  MoveL 3325 to (-39.23, 44.12, 59.84) mm, rotated rx -180 ry 0 rz 180 deg; joints [-136.898, -56.439, -94.12, 47.06, 68.969, -21.09]
  MoveL 3326 to (-39.23, 44.12, 59.84) mm, rotated rx -180 ry 0 rz 180 deg; joints [-136.898, -56.439, -94.12, 47.06, 68.969, -21.09]
  Call Extruder(64.50294)
  MoveL 3327 to (-39.1, 43.83, 59.84) mm, rotated rx 180 ry 0 rz -180 deg; joints [-136.946, -56.434, -94.139, 47.008, 68.961, -21.062]
  MoveL 3328 to (-39.1, 43.83, 59.84) mm, rotated rx 180 ry 0 rz -180 deg; joints [-136.946, -56.434, -94.139, 47.008, 68.961, -21.062]
  Call Extruder(64.66063)
  MoveL 3329 to (-39, 43.58, 59.84) mm, rotated rx -180 ry 0 rz -180 deg; joints [-136.988, -56.429, -94.155, 46.963, 68.953, -21.038]
  MoveL 3330 to (-39, 43.58, 59.84) mm, rotated rx -180 ry 0 rz -180 deg; joints [-136.988, -56.429, -94.155, 46.963, 68.953, -21.038]
  Call Extruder(64.81891)
  MoveL 3331 to (-38.89, 43.34, 59.84) mm, rotated rx 180 ry 0 rz 180 deg; joints [-137.029, -56.425, -94.17, 46.919, 68.946, -21.015]
  MoveL 3332 to (-38.89, 43.34, 59.84) mm, rotated rx 180 ry 0 rz 180 deg; joints [-137.029, -56.425, -94.17, 46.919, 68.946, -21.015]
  Call Extruder(65.00094)
  MoveL 3333 to (-38.75, 43.06, 59.84) mm, rotated rx 180 ry 0 rz -180 deg; joints [-137.078, -56.421, -94.184, 46.867, 68.935, -20.989]
  MoveL 3334 to (-38.75, 43.06, 59.84) mm, rotated rx 180 ry 0 rz -180 deg; joints [-137.078, -56.421, -94.184, 46.867, 68.935, -20.989]
  Call Extruder(65.20749)
  MoveL 3335 to (-38.57, 42.75, 59.84) mm, rotated rx -180 ry 0 rz -180 deg; joints [-137.135, -56.417, -94.197, 46.808, 68.921, -20.961]
  MoveL 3336 to (-38.57, 42.75, 59.84) mm, rotated rx -180 ry 0 rz -180 deg; joints [-137.135, -56.417, -94.197, 46.808, 68.921, -20.961]
  Call Extruder(65.41482)
  MoveL 3337 to (-38.4, 42.45, 59.84) mm, rotated rx 180 ry 0 rz -180 deg; joints [-137.191, -56.413, -94.21, 46.749, 68.908, -20.934]
  MoveL 3338 to (-38.4, 42.45, 59.84) mm, rotated rx 180 ry 0 rz -180 deg; joints [-137.191, -56.413, -94.21, 46.749, 68.908, -20.934]
  Call Extruder(65.62294)
  MoveL 3339 to (-38.22, 42.15, 59.84) mm, rotated rx 180 ry 0 rz 180 deg; joints [-137.247, -56.41, -94.223, 46.69, 68.894, -20.906]
  MoveL 3340 to (-38.22, 42.15, 59.84) mm, rotated rx 180 ry 0 rz 180 deg; joints [-137.247, -56.41, -94.223, 46.69, 68.894, -20.906]
  Call Extruder(65.74065)
  MoveL 3341 to (-38.12, 41.97, 59.84) mm, rotated rx -180 ry 0 rz -180 deg; joints [-137.279, -56.408, -94.231, 46.657, 68.886, -20.891]
  MoveL 3342 to (-38.12, 41.97, 59.84) mm, rotated rx -180 ry 0 rz -180 deg; joints [-137.279, -56.408, -94.231, 46.657, 68.886, -20.891]
  Call Extruder(66.07350)
  MoveL 3343 to (-37.79, 41.52, 59.84) mm, rotated rx 180 ry 0 rz 180 deg; joints [-137.37, -56.405, -94.241, 46.564, 68.859, -20.852]
  MoveL 3344 to (-37.79, 41.52, 59.84) mm, rotated rx 180 ry 0 rz 180 deg; joints [-137.37, -56.405, -94.241, 46.564, 68.859, -20.852]
  Call Extruder(66.40753)
  MoveL 3345 to (-37.47, 41.07, 59.84) mm, rotated rx 180 ry 0 rz 180 deg; joints [-137.461, -56.402, -94.252, 46.47, 68.832, -20.813]
  MoveL 3346 to (-37.47, 41.07, 59.84) mm, rotated rx 180 ry 0 rz 180 deg; joints [-137.461, -56.402, -94.252, 46.47, 68.832, -20.813]
  Call Extruder(66.57512)
  MoveL 3347 to (-37.3, 40.85, 59.84) mm, rotated rx 180 ry 0 rz 180 deg; joints [-137.506, -56.4, -94.257, 46.424, 68.819, -20.794]
  Call Extruder(67.40443)
  MoveL 3348 to (-36.39, 39.81, 59.84) mm, rotated rx 180 ry 0 rz -180 deg; joints [-137.733, -56.399, -94.262, 46.195, 68.74, -20.709]
  Call Extruder(68.03550)
  MoveL 3349 to (-35.6, 39.11, 59.84) mm, rotated rx 180 ry 0 rz 180 deg; joints [-137.904, -56.404, -94.243, 46.027, 68.67, -20.657]
  MoveL 3350 to (-35.6, 39.11, 59.84) mm, rotated rx 180 ry 0 rz 180 deg; joints [-137.904, -56.404, -94.243, 46.027, 68.67, -20.657]
  Call Extruder(68.23307)
  MoveL 3351 to (-35.35, 38.9, 59.84) mm, rotated rx 180 ry 0 rz -180 deg; joints [-137.958, -56.406, -94.235, 45.974, 68.648, -20.641]
  Call Extruder(68.56709)
  MoveL 3352 to (-34.9, 38.57, 59.84) mm, rotated rx 180 ry 0 rz -180 deg; joints [-138.048, -56.412, -94.216, 45.888, 68.606, -20.619]
  MoveL 3353 to (-34.9, 38.57, 59.84) mm, rotated rx 180 ry 0 rz -180 deg; joints [-138.048, -56.412, -94.216, 45.888, 68.606, -20.619]
  Call Extruder(68.89992)
  MoveL 3354 to (-34.45, 38.24, 59.84) mm, rotated rx -180 ry 0 rz 180 deg; joints [-138.137, -56.417, -94.196, 45.802, 68.565, -20.597]
  MoveL 3355 to (-34.45, 38.24, 59.84) mm, rotated rx -180 ry 0 rz 180 deg; joints [-138.137, -56.417, -94.196, 45.802, 68.565, -20.597]
  Call Extruder(69.07917)
  MoveL 3356 to (-34.21, 38.07, 59.84) mm, rotated rx 180 ry 0 rz 180 deg; joints [-138.185, -56.42, -94.185, 45.756, 68.543, -20.586]
  MoveL 3357 to (-34.21, 38.07, 59.84) mm, rotated rx 180 ry 0 rz 180 deg; joints [-138.185, -56.42, -94.185, 45.756, 68.543, -20.586]
  Call Extruder(69.28728)
  MoveL 3358 to (-33.9, 37.89, 59.84) mm, rotated rx 180 ry 0 rz -180 deg; joints [-138.24, -56.426, -94.167, 45.705, 68.514, -20.576]
  MoveL 3359 to (-33.9, 37.89, 59.84) mm, rotated rx 180 ry 0 rz -180 deg; joints [-138.24, -56.426, -94.167, 45.705, 68.514, -20.576]
  Call Extruder(69.49461)
  MoveL 3360 to (-33.6, 37.71, 59.84) mm, rotated rx -180 ry 0 rz -180 deg; joints [-138.295, -56.431, -94.149, 45.653, 68.486, -20.566]
  MoveL 3361 to (-33.6, 37.71, 59.84) mm, rotated rx -180 ry 0 rz -180 deg; joints [-138.295, -56.431, -94.149, 45.653, 68.486, -20.566]
  Call Extruder(69.70116)
  MoveL 3362 to (-33.29, 37.54, 59.84) mm, rotated rx 180 ry 0 rz 180 deg; joints [-138.349, -56.436, -94.13, 45.602, 68.458, -20.556]
  MoveL 3363 to (-33.29, 37.54, 59.84) mm, rotated rx 180 ry 0 rz 180 deg; joints [-138.349, -56.436, -94.13, 45.602, 68.458, -20.556]
  Call Extruder(69.90693)
  MoveL 3364 to (-32.99, 37.36, 59.84) mm, rotated rx 180 ry 0 rz 180 deg; joints [-138.404, -56.441, -94.112, 45.551, 68.429, -20.546]
  MoveL 3365 to (-32.99, 37.36, 59.84) mm, rotated rx 180 ry 0 rz 180 deg; joints [-138.404, -56.441, -94.112, 45.551, 68.429, -20.546]
  Call Extruder(70.06523)
  MoveL 3366 to (-32.74, 37.26, 59.84) mm, rotated rx -180 ry 0 rz 180 deg; joints [-138.444, -56.447, -94.092, 45.514, 68.405, -20.541]
  MoveL 3367 to (-32.74, 37.26, 59.84) mm, rotated rx -180 ry 0 rz 180 deg; joints [-138.444, -56.447, -94.092, 45.514, 68.405, -20.541]
  Call Extruder(70.22293)
  MoveL 3368 to (-32.49, 37.15, 59.84) mm, rotated rx 180 ry 0 rz 180 deg; joints [-138.484, -56.452, -94.073, 45.478, 68.381, -20.537]
  MoveL 3369 to (-32.49, 37.15, 59.84) mm, rotated rx 180 ry 0 rz 180 deg; joints [-138.484, -56.452, -94.073, 45.478, 68.381, -20.537]
  Call Extruder(70.39301)
  MoveL 3370 to (-32.22, 37.03, 59.84) mm, rotated rx -180 ry 0 rz 180 deg; joints [-138.527, -56.459, -94.051, 45.439, 68.356, -20.533]
  MoveL 3371 to (-32.22, 37.03, 59.84) mm, rotated rx -180 ry 0 rz 180 deg; joints [-138.527, -56.459, -94.051, 45.439, 68.356, -20.533]
  Call Extruder(70.57535)
  MoveL 3372 to (-31.93, 36.91, 59.84) mm, rotated rx 180 ry 0 rz 180 deg; joints [-138.574, -56.465, -94.028, 45.397, 68.328, -20.528]
  MoveL 3373 to (-31.93, 36.91, 59.84) mm, rotated rx 180 ry 0 rz 180 deg; joints [-138.574, -56.465, -94.028, 45.397, 68.328, -20.528]
  Call Extruder(70.75693)
  MoveL 3374 to (-31.64, 36.79, 59.84) mm, rotated rx 180 ry 0 rz 180 deg; joints [-138.62, -56.472, -94.005, 45.355, 68.3, -20.524]
  MoveL 3375 to (-31.64, 36.79, 59.84) mm, rotated rx 180 ry 0 rz 180 deg; joints [-138.62, -56.472, -94.005, 45.355, 68.3, -20.524]
  Call Extruder(70.85628)
  MoveL 3376 to (-31.47, 36.74, 59.84) mm, rotated rx 180 ry 0 rz -180 deg; joints [-138.645, -56.476, -93.99, 45.333, 68.284, -20.523]
  MoveL 3377 to (-31.47, 36.74, 59.84) mm, rotated rx 180 ry 0 rz -180 deg; joints [-138.645, -56.476, -93.99, 45.333, 68.284, -20.523]
  Call Extruder(70.95529)
  MoveL 3378 to (-31.31, 36.69, 59.84) mm, rotated rx 180 ry 0 rz 180 deg; joints [-138.669, -56.48, -93.975, 45.311, 68.268, -20.522]
  MoveL 3379 to (-31.31, 36.69, 59.84) mm, rotated rx 180 ry 0 rz 180 deg; joints [-138.669, -56.48, -93.975, 45.311, 68.268, -20.522]
  Call Extruder(71.05746)
  MoveL 3380 to (-31.14, 36.63, 59.84) mm, rotated rx -180 ry 0 rz 180 deg; joints [-138.694, -56.485, -93.96, 45.289, 68.251, -20.521]
  MoveL 3381 to (-31.14, 36.63, 59.84) mm, rotated rx -180 ry 0 rz 180 deg; joints [-138.694, -56.485, -93.96, 45.289, 68.251, -20.521]
  Call Extruder(71.16269)
  MoveL 3382 to (-30.96, 36.57, 59.84) mm, rotated rx 180 ry 0 rz -180 deg; joints [-138.72, -56.489, -93.944, 45.266, 68.234, -20.52]
  MoveL 3383 to (-30.96, 36.57, 59.84) mm, rotated rx 180 ry 0 rz -180 deg; joints [-138.72, -56.489, -93.944, 45.266, 68.234, -20.52]
  Call Extruder(71.26752)
  MoveL 3384 to (-30.78, 36.52, 59.84) mm, rotated rx 180 ry 0 rz -180 deg; joints [-138.746, -56.494, -93.928, 45.243, 68.217, -20.519]
  MoveL 3385 to (-30.78, 36.52, 59.84) mm, rotated rx 180 ry 0 rz -180 deg; joints [-138.746, -56.494, -93.928, 45.243, 68.217, -20.519]
  Call Extruder(71.38542)
  MoveL 3386 to (-30.58, 36.45, 59.84) mm, rotated rx 180 ry 0 rz 180 deg; joints [-138.776, -56.499, -93.909, 45.217, 68.197, -20.518]
  MoveL 3387 to (-30.58, 36.45, 59.84) mm, rotated rx 180 ry 0 rz 180 deg; joints [-138.776, -56.499, -93.909, 45.217, 68.197, -20.518]
  Call Extruder(71.51620)
  MoveL 3388 to (-30.36, 36.38, 59.84) mm, rotated rx -180 ry 0 rz 180 deg; joints [-138.808, -56.505, -93.889, 45.189, 68.175, -20.517]
  MoveL 3389 to (-30.36, 36.38, 59.84) mm, rotated rx -180 ry 0 rz 180 deg; joints [-138.808, -56.505, -93.889, 45.189, 68.175, -20.517]
  Call Extruder(71.64643)
  MoveL 3390 to (-30.14, 36.32, 59.84) mm, rotated rx 180 ry 0 rz 180 deg; joints [-138.84, -56.511, -93.868, 45.16, 68.154, -20.516]
  MoveL 3391 to (-30.14, 36.32, 59.84) mm, rotated rx 180 ry 0 rz 180 deg; joints [-138.84, -56.511, -93.868, 45.16, 68.154, -20.516]
  Call Extruder(71.77608)
  MoveL 3392 to (-29.91, 36.25, 59.84) mm, rotated rx 180 ry 0 rz -180 deg; joints [-138.873, -56.517, -93.847, 45.132, 68.132, -20.516]
  MoveL 3393 to (-29.91, 36.25, 59.84) mm, rotated rx 180 ry 0 rz -180 deg; joints [-138.873, -56.517, -93.847, 45.132, 68.132, -20.516]
  Call Extruder(71.90518)
  MoveL 3394 to (-29.69, 36.18, 59.84) mm, rotated rx -180 ry 0 rz -180 deg; joints [-138.905, -56.523, -93.826, 45.104, 68.11, -20.515]
  MoveL 3395 to (-29.69, 36.18, 59.84) mm, rotated rx -180 ry 0 rz -180 deg; joints [-138.905, -56.523, -93.826, 45.104, 68.11, -20.515]
  Call Extruder(72.02025)
  MoveL 3396 to (-29.48, 36.14, 59.84) mm, rotated rx -180 ry 0 rz 180 deg; joints [-138.932, -56.529, -93.805, 45.08, 68.09, -20.516]
  MoveL 3397 to (-29.48, 36.14, 59.84) mm, rotated rx -180 ry 0 rz 180 deg; joints [-138.932, -56.529, -93.805, 45.08, 68.09, -20.516]
  Call Extruder(72.13487)
  MoveL 3398 to (-29.28, 36.09, 59.84) mm, rotated rx -180 ry 0 rz 180 deg; joints [-138.96, -56.535, -93.784, 45.057, 68.07, -20.517]
  MoveL 3399 to (-29.28, 36.09, 59.84) mm, rotated rx -180 ry 0 rz 180 deg; joints [-138.96, -56.535, -93.784, 45.057, 68.07, -20.517]
  Call Extruder(72.24904)
  MoveL 3400 to (-29.08, 36.05, 59.84) mm, rotated rx 180 ry 0 rz -180 deg; joints [-138.987, -56.541, -93.763, 45.034, 68.049, -20.518]
  MoveL 3401 to (-29.08, 36.05, 59.84) mm, rotated rx 180 ry 0 rz -180 deg; joints [-138.987, -56.541, -93.763, 45.034, 68.049, -20.518]
  Call Extruder(72.36276)
  MoveL 3402 to (-28.87, 36, 59.84) mm, rotated rx 180 ry 0 rz -180 deg; joints [-139.014, -56.547, -93.742, 45.01, 68.029, -20.519]
  MoveL 3403 to (-28.87, 36, 59.84) mm, rotated rx 180 ry 0 rz -180 deg; joints [-139.014, -56.547, -93.742, 45.01, 68.029, -20.519]
  Call Extruder(72.48818)
  MoveL 3404 to (-28.64, 35.96, 59.84) mm, rotated rx 180 ry 0 rz 180 deg; joints [-139.044, -56.554, -93.719, 44.985, 68.007, -20.521]
  MoveL 3405 to (-28.64, 35.96, 59.84) mm, rotated rx 180 ry 0 rz 180 deg; joints [-139.044, -56.554, -93.719, 44.985, 68.007, -20.521]
  Call Extruder(72.62516)
  MoveL 3406 to (-28.4, 35.91, 59.84) mm, rotated rx 180 ry 0 rz -180 deg; joints [-139.077, -56.561, -93.692, 44.957, 67.982, -20.523]
  MoveL 3407 to (-28.4, 35.91, 59.84) mm, rotated rx 180 ry 0 rz -180 deg; joints [-139.077, -56.561, -93.692, 44.957, 67.982, -20.523]
  Call Extruder(72.76152)
  MoveL 3408 to (-28.15, 35.86, 59.84) mm, rotated rx -180 ry 0 rz 180 deg; joints [-139.109, -56.569, -93.666, 44.93, 67.958, -20.525]
  MoveL 3409 to (-28.15, 35.86, 59.84) mm, rotated rx -180 ry 0 rz 180 deg; joints [-139.109, -56.569, -93.666, 44.93, 67.958, -20.525]
  Call Extruder(72.89728)
  MoveL 3410 to (-27.9, 35.81, 59.84) mm, rotated rx 180 ry 0 rz 180 deg; joints [-139.142, -56.576, -93.64, 44.902, 67.933, -20.526]
  MoveL 3411 to (-27.9, 35.81, 59.84) mm, rotated rx 180 ry 0 rz 180 deg; joints [-139.142, -56.576, -93.64, 44.902, 67.933, -20.526]
  Call Extruder(73.03243)
  MoveL 3412 to (-27.65, 35.76, 59.84) mm, rotated rx -180 ry 0 rz 180 deg; joints [-139.174, -56.584, -93.613, 44.875, 67.908, -20.528]
  MoveL 3413 to (-27.65, 35.76, 59.84) mm, rotated rx -180 ry 0 rz 180 deg; joints [-139.174, -56.584, -93.613, 44.875, 67.908, -20.528]
  Call Extruder(73.16696)
  MoveL 3414 to (-27.4, 35.71, 59.84) mm, rotated rx 180 ry 0 rz 180 deg; joints [-139.207, -56.591, -93.587, 44.847, 67.884, -20.53]
  MoveL 3415 to (-27.4, 35.71, 59.84) mm, rotated rx 180 ry 0 rz 180 deg; joints [-139.207, -56.591, -93.587, 44.847, 67.884, -20.53]
  Call Extruder(73.30089)
  MoveL 3416 to (-27.15, 35.66, 59.84) mm, rotated rx 180 ry 0 rz 180 deg; joints [-139.239, -56.599, -93.561, 44.82, 67.859, -20.532]
  MoveL 3417 to (-27.15, 35.66, 59.84) mm, rotated rx 180 ry 0 rz 180 deg; joints [-139.239, -56.599, -93.561, 44.82, 67.859, -20.532]
  Call Extruder(73.44875)
  MoveL 3418 to (-26.87, 35.61, 59.84) mm, rotated rx 180 ry 0 rz -180 deg; joints [-139.275, -56.608, -93.531, 44.79, 67.831, -20.535]
  MoveL 3419 to (-26.87, 35.61, 59.84) mm, rotated rx 180 ry 0 rz -180 deg; joints [-139.275, -56.608, -93.531, 44.79, 67.831, -20.535]
  Call Extruder(73.61048)
  MoveL 3420 to (-26.57, 35.56, 59.84) mm, rotated rx 180 ry 0 rz -180 deg; joints [-139.313, -56.617, -93.497, 44.758, 67.801, -20.539]
  MoveL 3421 to (-26.57, 35.56, 59.84) mm, rotated rx 180 ry 0 rz -180 deg; joints [-139.313, -56.617, -93.497, 44.758, 67.801, -20.539]
  Call Extruder(73.77149)
  MoveL 3422 to (-26.26, 35.51, 59.84) mm, rotated rx 180 ry 0 rz 180 deg; joints [-139.351, -56.627, -93.463, 44.727, 67.77, -20.542]
  MoveL 3423 to (-26.26, 35.51, 59.84) mm, rotated rx 180 ry 0 rz 180 deg; joints [-139.351, -56.627, -93.463, 44.727, 67.77, -20.542]
  Call Extruder(73.93177)
  MoveL 3424 to (-25.96, 35.46, 59.84) mm, rotated rx 180 ry 0 rz 180 deg; joints [-139.39, -56.637, -93.43, 44.695, 67.74, -20.546]
  MoveL 3425 to (-25.96, 35.46, 59.84) mm, rotated rx 180 ry 0 rz 180 deg; joints [-139.39, -56.637, -93.43, 44.695, 67.74, -20.546]
  Call Extruder(74.09132)
  MoveL 3426 to (-25.65, 35.42, 59.84) mm, rotated rx 180 ry 0 rz 180 deg; joints [-139.428, -56.647, -93.396, 44.663, 67.709, -20.55]
  MoveL 3427 to (-25.65, 35.42, 59.84) mm, rotated rx 180 ry 0 rz 180 deg; joints [-139.428, -56.647, -93.396, 44.663, 67.709, -20.55]
  Call Extruder(74.25014)
  MoveL 3428 to (-25.34, 35.37, 59.84) mm, rotated rx 180 ry 0 rz 180 deg; joints [-139.466, -56.657, -93.362, 44.631, 67.679, -20.553]
  MoveL 3429 to (-25.34, 35.37, 59.84) mm, rotated rx 180 ry 0 rz 180 deg; joints [-139.466, -56.657, -93.362, 44.631, 67.679, -20.553]
  Call Extruder(74.42881)
  MoveL 3430 to (-25, 35.32, 59.84) mm, rotated rx 180 ry 0 rz -180 deg; joints [-139.508, -56.668, -93.322, 44.597, 67.644, -20.558]
  MoveL 3431 to (-25, 35.32, 59.84) mm, rotated rx 180 ry 0 rz -180 deg; joints [-139.508, -56.668, -93.322, 44.597, 67.644, -20.558]
  Call Extruder(74.62725)
  MoveL 3432 to (-24.61, 35.27, 59.84) mm, rotated rx 180 ry 0 rz 180 deg; joints [-139.554, -56.681, -93.278, 44.559, 67.605, -20.564]
  MoveL 3433 to (-24.61, 35.27, 59.84) mm, rotated rx 180 ry 0 rz 180 deg; joints [-139.554, -56.681, -93.278, 44.559, 67.605, -20.564]
  Call Extruder(74.82483)
  MoveL 3434 to (-24.22, 35.23, 59.84) mm, rotated rx 180 ry 0 rz -180 deg; joints [-139.6, -56.694, -93.233, 44.522, 67.566, -20.571]
  MoveL 3435 to (-24.22, 35.23, 59.84) mm, rotated rx 180 ry 0 rz -180 deg; joints [-139.6, -56.694, -93.233, 44.522, 67.566, -20.571]
  Call Extruder(75.02153)
  MoveL 3436 to (-23.83, 35.18, 59.84) mm, rotated rx 180 ry 0 rz 180 deg; joints [-139.647, -56.707, -93.188, 44.484, 67.527, -20.577]
  MoveL 3437 to (-23.83, 35.18, 59.84) mm, rotated rx 180 ry 0 rz 180 deg; joints [-139.647, -56.707, -93.188, 44.484, 67.527, -20.577]
  Call Extruder(75.21737)
  MoveL 3438 to (-23.45, 35.14, 59.84) mm, rotated rx 180 ry 0 rz 180 deg; joints [-139.693, -56.72, -93.143, 44.447, 67.488, -20.583]
  MoveL 3439 to (-23.45, 35.14, 59.84) mm, rotated rx 180 ry 0 rz 180 deg; joints [-139.693, -56.72, -93.143, 44.447, 67.488, -20.583]
  Call Extruder(75.51277)
  MoveL 3440 to (-22.86, 35.09, 59.84) mm, rotated rx -180 ry 0 rz 180 deg; joints [-139.76, -56.741, -93.072, 44.393, 67.429, -20.595]
  MoveL 3441 to (-22.86, 35.09, 59.84) mm, rotated rx -180 ry 0 rz 180 deg; joints [-139.76, -56.741, -93.072, 44.393, 67.429, -20.595]
  Call Extruder(75.80683)
  MoveL 3442 to (-22.27, 35.04, 59.84) mm, rotated rx -180 ry 0 rz -180 deg; joints [-139.826, -56.762, -93.001, 44.34, 67.369, -20.608]
  MoveL 3443 to (-22.27, 35.04, 59.84) mm, rotated rx -180 ry 0 rz -180 deg; joints [-139.826, -56.762, -93.001, 44.34, 67.369, -20.608]
  Call Extruder(76.09956)
  MoveL 3444 to (-21.68, 35, 59.84) mm, rotated rx -180 ry 0 rz -180 deg; joints [-139.893, -56.783, -92.929, 44.287, 67.31, -20.62]
  MoveL 3445 to (-21.68, 35, 59.84) mm, rotated rx -180 ry 0 rz -180 deg; joints [-139.893, -56.783, -92.929, 44.287, 67.31, -20.62]
  Call Extruder(76.67301)
  MoveL 3446 to (-20.52, 34.95, 59.84) mm, rotated rx 180 ry 0 rz -180 deg; joints [-140.019, -56.825, -92.783, 44.19, 67.192, -20.648]
  MoveL 3447 to (-20.52, 34.95, 59.84) mm, rotated rx 180 ry 0 rz -180 deg; joints [-140.019, -56.825, -92.783, 44.19, 67.192, -20.648]
  Call Extruder(77.38698)
  MoveL 3448 to (-19.06, 34.91, 59.84) mm, rotated rx 180 ry 0 rz 180 deg; joints [-140.173, -56.88, -92.598, 44.072, 67.043, -20.686]
  Call Extruder(194.23372)
  MoveL 3449 to (219.06, 34.91, 59.84) mm, rotated rx 180 ry 0 rz 180 deg; joints [-155.896, -73.502, -50.043, 38.995, 40.467, -31.631]
  Call Extruder(194.66228)
  MoveL 3450 to (219.94, 34.93, 59.84) mm, rotated rx 180 ry 0 rz -180 deg; joints [-155.931, -73.601, -49.824, 39.038, 40.355, -31.714]
  MoveL 3451 to (219.94, 34.93, 59.84) mm, rotated rx 180 ry 0 rz -180 deg; joints [-155.931, -73.601, -49.824, 39.038, 40.355, -31.714]
  Call Extruder(195.23572)
  MoveL 3452 to (221.1, 34.97, 59.84) mm, rotated rx 180 ry 0 rz 180 deg; joints [-155.975, -73.734, -49.529, 39.101, 40.206, -31.827]
  MoveL 3453 to (221.1, 34.97, 59.84) mm, rotated rx 180 ry 0 rz 180 deg; joints [-155.975, -73.734, -49.529, 39.101, 40.206, -31.827]
  Call Extruder(195.67004)
  MoveL 3454 to (221.97, 35.02, 59.84) mm, rotated rx 180 ry 0 rz 180 deg; joints [-156.007, -73.836, -49.304, 39.151, 40.094, -31.916]
  MoveL 3455 to (221.97, 35.02, 59.84) mm, rotated rx 180 ry 0 rz 180 deg; joints [-156.007, -73.836, -49.304, 39.151, 40.094, -31.916]
  Call Extruder(195.96409)
  MoveL 3456 to (222.56, 35.07, 59.84) mm, rotated rx 180 ry 0 rz -180 deg; joints [-156.027, -73.905, -49.15, 39.188, 40.018, -31.978]
  MoveL 3457 to (222.56, 35.07, 59.84) mm, rotated rx 180 ry 0 rz -180 deg; joints [-156.027, -73.905, -49.15, 39.188, 40.018, -31.978]
  Call Extruder(196.25948)
  MoveL 3458 to (223.15, 35.11, 59.84) mm, rotated rx 180 ry 0 rz 180 deg; joints [-156.047, -73.975, -48.997, 39.225, 39.943, -32.04]
  MoveL 3459 to (223.15, 35.11, 59.84) mm, rotated rx 180 ry 0 rz 180 deg; joints [-156.047, -73.975, -48.997, 39.225, 39.943, -32.04]
  Call Extruder(196.50572)
  MoveL 3460 to (223.64, 35.16, 59.84) mm, rotated rx 180 ry 0 rz 180 deg; joints [-156.062, -74.033, -48.868, 39.257, 39.88, -32.094]
  MoveL 3461 to (223.64, 35.16, 59.84) mm, rotated rx 180 ry 0 rz 180 deg; joints [-156.062, -74.033, -48.868, 39.257, 39.88, -32.094]
  Call Extruder(196.70242)
  MoveL 3462 to (224.03, 35.21, 59.84) mm, rotated rx -180 ry 0 rz 180 deg; joints [-156.074, -74.08, -48.765, 39.285, 39.83, -32.138]
  MoveL 3463 to (224.03, 35.21, 59.84) mm, rotated rx -180 ry 0 rz 180 deg; joints [-156.074, -74.08, -48.765, 39.285, 39.83, -32.138]
  Call Extruder(196.90000)
  MoveL 3464 to (224.42, 35.25, 59.84) mm, rotated rx 180 ry 0 rz 180 deg; joints [-156.086, -74.127, -48.661, 39.312, 39.78, -32.182]
  MoveL 3465 to (224.42, 35.25, 59.84) mm, rotated rx 180 ry 0 rz 180 deg; joints [-156.086, -74.127, -48.661, 39.312, 39.78, -32.182]
  Call Extruder(197.09844)
  MoveL 3466 to (224.8, 35.3, 59.84) mm, rotated rx -180 ry 0 rz 180 deg; joints [-156.097, -74.174, -48.558, 39.34, 39.73, -32.226]
  MoveL 3467 to (224.8, 35.3, 59.84) mm, rotated rx -180 ry 0 rz 180 deg; joints [-156.097, -74.174, -48.558, 39.34, 39.73, -32.226]
  Call Extruder(197.29775)
  MoveL 3468 to (225.19, 35.34, 59.84) mm, rotated rx -180 ry 0 rz 180 deg; joints [-156.109, -74.221, -48.454, 39.368, 39.68, -32.27]
  MoveL 3469 to (225.19, 35.34, 59.84) mm, rotated rx -180 ry 0 rz 180 deg; joints [-156.109, -74.221, -48.454, 39.368, 39.68, -32.27]
  Call Extruder(197.45657)
  MoveL 3470 to (225.5, 35.39, 59.84) mm, rotated rx 180 ry 0 rz 180 deg; joints [-156.117, -74.259, -48.371, 39.392, 39.641, -32.307]
  MoveL 3471 to (225.5, 35.39, 59.84) mm, rotated rx 180 ry 0 rz 180 deg; joints [-156.117, -74.259, -48.371, 39.392, 39.641, -32.307]
  Call Extruder(197.61612)
  MoveL 3472 to (225.8, 35.44, 59.84) mm, rotated rx 180 ry 0 rz 180 deg; joints [-156.125, -74.297, -48.287, 39.416, 39.601, -32.345]
  MoveL 3473 to (225.8, 35.44, 59.84) mm, rotated rx 180 ry 0 rz 180 deg; joints [-156.125, -74.297, -48.287, 39.416, 39.601, -32.345]
  Call Extruder(197.77640)
  MoveL 3474 to (226.11, 35.49, 59.84) mm, rotated rx 180 ry 0 rz -180 deg; joints [-156.133, -74.335, -48.204, 39.441, 39.562, -32.382]
  MoveL 3475 to (226.11, 35.49, 59.84) mm, rotated rx 180 ry 0 rz -180 deg; joints [-156.133, -74.335, -48.204, 39.441, 39.562, -32.382]
  Call Extruder(197.93740)
  MoveL 3476 to (226.41, 35.54, 59.84) mm, rotated rx 180 ry 0 rz -180 deg; joints [-156.141, -74.373, -48.12, 39.465, 39.522, -32.419]
  MoveL 3477 to (226.41, 35.54, 59.84) mm, rotated rx 180 ry 0 rz -180 deg; joints [-156.141, -74.373, -48.12, 39.465, 39.522, -32.419]
  Call Extruder(198.09914)
  MoveL 3478 to (226.72, 35.59, 59.84) mm, rotated rx 180 ry 0 rz 180 deg; joints [-156.149, -74.411, -48.036, 39.49, 39.483, -32.457]
  MoveL 3479 to (226.72, 35.59, 59.84) mm, rotated rx 180 ry 0 rz 180 deg; joints [-156.149, -74.411, -48.036, 39.49, 39.483, -32.457]
  Call Extruder(198.26160)
  MoveL 3480 to (227.03, 35.63, 59.84) mm, rotated rx -180 ry 0 rz 180 deg; joints [-156.157, -74.449, -47.952, 39.515, 39.443, -32.494]
  MoveL 3481 to (227.03, 35.63, 59.84) mm, rotated rx -180 ry 0 rz 180 deg; joints [-156.157, -74.449, -47.952, 39.515, 39.443, -32.494]
  Call Extruder(198.39552)
  MoveL 3482 to (227.27, 35.68, 59.84) mm, rotated rx 180 ry 0 rz 180 deg; joints [-156.162, -74.481, -47.883, 39.537, 39.411, -32.527]
  MoveL 3483 to (227.27, 35.68, 59.84) mm, rotated rx 180 ry 0 rz 180 deg; joints [-156.162, -74.481, -47.883, 39.537, 39.411, -32.527]
  Call Extruder(198.53006)
  MoveL 3484 to (227.52, 35.73, 59.84) mm, rotated rx -180 ry 0 rz 180 deg; joints [-156.168, -74.513, -47.813, 39.559, 39.379, -32.559]
  MoveL 3485 to (227.52, 35.73, 59.84) mm, rotated rx -180 ry 0 rz 180 deg; joints [-156.168, -74.513, -47.813, 39.559, 39.379, -32.559]
  Call Extruder(198.66521)
  MoveL 3486 to (227.77, 35.78, 59.84) mm, rotated rx -180 ry 0 rz -180 deg; joints [-156.173, -74.545, -47.743, 39.581, 39.346, -32.591]
  MoveL 3487 to (227.77, 35.78, 59.84) mm, rotated rx -180 ry 0 rz -180 deg; joints [-156.173, -74.545, -47.743, 39.581, 39.346, -32.591]
  Call Extruder(198.80097)
  MoveL 3488 to (228.02, 35.83, 59.84) mm, rotated rx 180 ry 0 rz 180 deg; joints [-156.179, -74.576, -47.673, 39.603, 39.314, -32.624]
  MoveL 3489 to (228.02, 35.83, 59.84) mm, rotated rx 180 ry 0 rz 180 deg; joints [-156.179, -74.576, -47.673, 39.603, 39.314, -32.624]
  Call Extruder(198.93734)
  MoveL 3490 to (228.27, 35.88, 59.84) mm, rotated rx 180 ry 0 rz -180 deg; joints [-156.185, -74.608, -47.603, 39.625, 39.282, -32.657]
  MoveL 3491 to (228.27, 35.88, 59.84) mm, rotated rx 180 ry 0 rz -180 deg; joints [-156.185, -74.608, -47.603, 39.625, 39.282, -32.657]
  Call Extruder(199.07431)
  MoveL 3492 to (228.52, 35.93, 59.84) mm, rotated rx 180 ry 0 rz 180 deg; joints [-156.19, -74.64, -47.534, 39.648, 39.25, -32.689]
  MoveL 3493 to (228.52, 35.93, 59.84) mm, rotated rx 180 ry 0 rz 180 deg; joints [-156.19, -74.64, -47.534, 39.648, 39.25, -32.689]
  Call Extruder(199.21190)
  MoveL 3494 to (228.77, 35.98, 59.84) mm, rotated rx 180 ry 0 rz 180 deg; joints [-156.196, -74.672, -47.463, 39.67, 39.217, -32.722]
  MoveL 3495 to (228.77, 35.98, 59.84) mm, rotated rx 180 ry 0 rz 180 deg; joints [-156.196, -74.672, -47.463, 39.67, 39.217, -32.722]
  Call Extruder(199.32562)
  MoveL 3496 to (228.97, 36.03, 59.84) mm, rotated rx 180 ry 0 rz 180 deg; joints [-156.2, -74.699, -47.405, 39.689, 39.191, -32.75]
  MoveL 3497 to (228.97, 36.03, 59.84) mm, rotated rx 180 ry 0 rz 180 deg; joints [-156.2, -74.699, -47.405, 39.689, 39.191, -32.75]
  Call Extruder(199.43979)
  MoveL 3498 to (229.18, 36.07, 59.84) mm, rotated rx 180 ry 0 rz 180 deg; joints [-156.204, -74.725, -47.347, 39.708, 39.164, -32.777]
  MoveL 3499 to (229.18, 36.07, 59.84) mm, rotated rx 180 ry 0 rz 180 deg; joints [-156.204, -74.725, -47.347, 39.708, 39.164, -32.777]
  Call Extruder(199.55441)
  MoveL 3500 to (229.38, 36.12, 59.84) mm, rotated rx 180 ry 0 rz -180 deg; joints [-156.208, -74.752, -47.289, 39.728, 39.138, -32.805]
  MoveL 3501 to (229.38, 36.12, 59.84) mm, rotated rx 180 ry 0 rz -180 deg; joints [-156.208, -74.752, -47.289, 39.728, 39.138, -32.805]
  Call Extruder(199.66948)
  MoveL 3502 to (229.59, 36.16, 59.84) mm, rotated rx 180 ry 0 rz 180 deg; joints [-156.212, -74.778, -47.231, 39.747, 39.111, -32.832]
  MoveL 3503 to (229.59, 36.16, 59.84) mm, rotated rx 180 ry 0 rz 180 deg; joints [-156.212, -74.778, -47.231, 39.747, 39.111, -32.832]
  Call Extruder(199.79172)
  MoveL 3504 to (229.8, 36.22, 59.84) mm, rotated rx 180 ry 0 rz 180 deg; joints [-156.216, -74.806, -47.169, 39.769, 39.083, -32.863]
  MoveL 3505 to (229.8, 36.22, 59.84) mm, rotated rx 180 ry 0 rz 180 deg; joints [-156.216, -74.806, -47.169, 39.769, 39.083, -32.863]
  Call Extruder(199.92138)
  MoveL 3506 to (230.02, 36.28, 59.84) mm, rotated rx 180 ry 0 rz -180 deg; joints [-156.219, -74.836, -47.103, 39.793, 39.054, -32.897]
  MoveL 3507 to (230.02, 36.28, 59.84) mm, rotated rx 180 ry 0 rz -180 deg; joints [-156.219, -74.836, -47.103, 39.793, 39.054, -32.897]
  Call Extruder(200.05161)
  MoveL 3508 to (230.25, 36.35, 59.84) mm, rotated rx 180 ry 0 rz 180 deg; joints [-156.221, -74.867, -47.038, 39.818, 39.025, -32.93]
  MoveL 3509 to (230.25, 36.35, 59.84) mm, rotated rx 180 ry 0 rz 180 deg; joints [-156.221, -74.867, -47.038, 39.818, 39.025, -32.93]
  Call Extruder(200.18241)
  MoveL 3510 to (230.47, 36.42, 59.84) mm, rotated rx 180 ry 0 rz -180 deg; joints [-156.224, -74.897, -46.971, 39.842, 38.996, -32.964]
  MoveL 3511 to (230.47, 36.42, 59.84) mm, rotated rx 180 ry 0 rz -180 deg; joints [-156.224, -74.897, -46.971, 39.842, 38.996, -32.964]
  Call Extruder(200.31377)
  MoveL 3512 to (230.69, 36.49, 59.84) mm, rotated rx 180 ry 0 rz 180 deg; joints [-156.227, -74.927, -46.905, 39.867, 38.967, -32.997]
  MoveL 3513 to (230.69, 36.49, 59.84) mm, rotated rx 180 ry 0 rz 180 deg; joints [-156.227, -74.927, -46.905, 39.867, 38.967, -32.997]
  Call Extruder(200.43194)
  MoveL 3514 to (230.89, 36.55, 59.84) mm, rotated rx 180 ry 0 rz 180 deg; joints [-156.229, -74.954, -46.846, 39.89, 38.941, -33.028]
  MoveL 3515 to (230.89, 36.55, 59.84) mm, rotated rx 180 ry 0 rz 180 deg; joints [-156.229, -74.954, -46.846, 39.89, 38.941, -33.028]
  Call Extruder(200.55059)
  MoveL 3516 to (231.09, 36.62, 59.84) mm, rotated rx -180 ry 0 rz 180 deg; joints [-156.231, -74.981, -46.786, 39.913, 38.915, -33.059]
  MoveL 3517 to (231.09, 36.62, 59.84) mm, rotated rx -180 ry 0 rz 180 deg; joints [-156.231, -74.981, -46.786, 39.913, 38.915, -33.059]
  Call Extruder(200.66975)
  MoveL 3518 to (231.29, 36.68, 59.84) mm, rotated rx 180 ry 0 rz 180 deg; joints [-156.233, -75.009, -46.727, 39.936, 38.889, -33.09]
  MoveL 3519 to (231.29, 36.68, 59.84) mm, rotated rx 180 ry 0 rz 180 deg; joints [-156.233, -75.009, -46.727, 39.936, 38.889, -33.09]
  Call Extruder(200.77883)
  MoveL 3520 to (231.47, 36.74, 59.84) mm, rotated rx 180 ry 0 rz 180 deg; joints [-156.235, -75.033, -46.673, 39.957, 38.866, -33.118]
  MoveL 3521 to (231.47, 36.74, 59.84) mm, rotated rx 180 ry 0 rz 180 deg; joints [-156.235, -75.033, -46.673, 39.957, 38.866, -33.118]
  Call Extruder(200.87772)
  MoveL 3522 to (231.64, 36.79, 59.84) mm, rotated rx 180 ry 0 rz 180 deg; joints [-156.237, -75.056, -46.624, 39.975, 38.844, -33.143]
  MoveL 3523 to (231.64, 36.79, 59.84) mm, rotated rx 180 ry 0 rz 180 deg; joints [-156.237, -75.056, -46.624, 39.975, 38.844, -33.143]
  Call Extruder(201.05968)
  MoveL 3524 to (231.93, 36.91, 59.84) mm, rotated rx 180 ry 0 rz 180 deg; joints [-156.238, -75.097, -46.533, 40.014, 38.806, -33.193]
  MoveL 3525 to (231.93, 36.91, 59.84) mm, rotated rx 180 ry 0 rz 180 deg; joints [-156.238, -75.097, -46.533, 40.014, 38.806, -33.193]
  Call Extruder(201.24239)
  MoveL 3526 to (232.22, 37.03, 59.84) mm, rotated rx 180 ry 0 rz 180 deg; joints [-156.238, -75.139, -46.442, 40.052, 38.768, -33.243]
  MoveL 3527 to (232.22, 37.03, 59.84) mm, rotated rx 180 ry 0 rz 180 deg; joints [-156.238, -75.139, -46.442, 40.052, 38.768, -33.243]
  Call Extruder(201.41281)
  MoveL 3528 to (232.49, 37.15, 59.84) mm, rotated rx 180 ry 0 rz 180 deg; joints [-156.239, -75.177, -46.358, 40.088, 38.733, -33.289]
  MoveL 3529 to (232.49, 37.15, 59.84) mm, rotated rx 180 ry 0 rz 180 deg; joints [-156.239, -75.177, -46.358, 40.088, 38.733, -33.289]
  Call Extruder(201.57081)
  MoveL 3530 to (232.74, 37.26, 59.84) mm, rotated rx 180 ry 0 rz 180 deg; joints [-156.239, -75.213, -46.28, 40.122, 38.701, -33.332]
  MoveL 3531 to (232.74, 37.26, 59.84) mm, rotated rx 180 ry 0 rz 180 deg; joints [-156.239, -75.213, -46.28, 40.122, 38.701, -33.332]
  Call Extruder(201.72941)
  MoveL 3532 to (232.99, 37.36, 59.84) mm, rotated rx -180 ry 0 rz -180 deg; joints [-156.239, -75.249, -46.202, 40.156, 38.668, -33.376]
  MoveL 3533 to (232.99, 37.36, 59.84) mm, rotated rx -180 ry 0 rz -180 deg; joints [-156.239, -75.249, -46.202, 40.156, 38.668, -33.376]
  Call Extruder(201.93558)
  MoveL 3534 to (233.29, 37.54, 59.84) mm, rotated rx 180 ry 0 rz 180 deg; joints [-156.236, -75.295, -46.101, 40.205, 38.628, -33.436]
  MoveL 3535 to (233.29, 37.54, 59.84) mm, rotated rx 180 ry 0 rz 180 deg; joints [-156.236, -75.295, -46.101, 40.205, 38.628, -33.436]
  Call Extruder(202.14252)
  MoveL 3536 to (233.6, 37.71, 59.84) mm, rotated rx 180 ry 0 rz 180 deg; joints [-156.232, -75.341, -46, 40.254, 38.589, -33.497]
  MoveL 3537 to (233.6, 37.71, 59.84) mm, rotated rx 180 ry 0 rz 180 deg; joints [-156.232, -75.341, -46, 40.254, 38.589, -33.497]
  Call Extruder(202.35025)
  MoveL 3538 to (233.9, 37.89, 59.84) mm, rotated rx 180 ry 0 rz 180 deg; joints [-156.228, -75.388, -45.899, 40.303, 38.549, -33.557]
  MoveL 3539 to (233.9, 37.89, 59.84) mm, rotated rx 180 ry 0 rz 180 deg; joints [-156.228, -75.388, -45.899, 40.303, 38.549, -33.557]
  Call Extruder(202.55875)
  MoveL 3540 to (234.21, 38.06, 59.84) mm, rotated rx -180 ry 0 rz 180 deg; joints [-156.224, -75.434, -45.798, 40.353, 38.509, -33.618]
  MoveL 3541 to (234.21, 38.06, 59.84) mm, rotated rx -180 ry 0 rz 180 deg; joints [-156.224, -75.434, -45.798, 40.353, 38.509, -33.618]
  Call Extruder(202.73829)
  MoveL 3542 to (234.45, 38.24, 59.84) mm, rotated rx -180 ry 0 rz 180 deg; joints [-156.218, -75.474, -45.712, 40.399, 38.478, -33.673]
  MoveL 3543 to (234.45, 38.24, 59.84) mm, rotated rx -180 ry 0 rz 180 deg; joints [-156.218, -75.474, -45.712, 40.399, 38.478, -33.673]
  Call Extruder(203.07171)
  MoveL 3544 to (234.9, 38.57, 59.84) mm, rotated rx -180 ry 0 rz -180 deg; joints [-156.206, -75.546, -45.553, 40.485, 38.419, -33.775]
  MoveL 3545 to (234.9, 38.57, 59.84) mm, rotated rx -180 ry 0 rz -180 deg; joints [-156.206, -75.546, -45.553, 40.485, 38.419, -33.775]
  Call Extruder(203.40631)
  MoveL 3546 to (235.35, 38.9, 59.84) mm, rotated rx 180 ry 0 rz 180 deg; joints [-156.195, -75.62, -45.394, 40.571, 38.36, -33.877]
  Call Extruder(204.23426)
  MoveL 3547 to (236.39, 39.81, 59.84) mm, rotated rx -180 ry 0 rz 180 deg; joints [-156.154, -75.797, -45.008, 40.798, 38.225, -34.139]
  Call Extruder(205.06220)
  MoveL 3548 to (237.3, 40.85, 59.84) mm, rotated rx 180 ry 0 rz 180 deg; joints [-156.097, -75.967, -44.638, 41.041, 38.106, -34.411]
  Call Extruder(205.22950)
  MoveL 3549 to (237.47, 41.07, 59.84) mm, rotated rx -180 ry 0 rz 180 deg; joints [-156.083, -76, -44.567, 41.091, 38.085, -34.466]
  MoveL 3550 to (237.47, 41.07, 59.84) mm, rotated rx -180 ry 0 rz 180 deg; joints [-156.083, -76, -44.567, 41.091, 38.085, -34.466]
  Call Extruder(205.56292)
  MoveL 3551 to (237.8, 41.52, 59.84) mm, rotated rx -180 ry 0 rz 180 deg; joints [-156.055, -76.066, -44.424, 41.193, 38.042, -34.578]
  MoveL 3552 to (237.8, 41.52, 59.84) mm, rotated rx -180 ry 0 rz 180 deg; joints [-156.055, -76.066, -44.424, 41.193, 38.042, -34.578]
  Call Extruder(205.89514)
  MoveL 3553 to (238.12, 41.98, 59.84) mm, rotated rx 180 ry 0 rz -180 deg; joints [-156.028, -76.133, -44.28, 41.295, 38, -34.689]
  MoveL 3554 to (238.12, 41.98, 59.84) mm, rotated rx 180 ry 0 rz -180 deg; joints [-156.028, -76.133, -44.28, 41.295, 38, -34.689]
  Call Extruder(206.01284)
  MoveL 3555 to (238.22, 42.15, 59.84) mm, rotated rx 180 ry 0 rz 180 deg; joints [-156.016, -76.155, -44.232, 41.332, 37.987, -34.729]
  MoveL 3556 to (238.22, 42.15, 59.84) mm, rotated rx 180 ry 0 rz 180 deg; joints [-156.016, -76.155, -44.232, 41.332, 37.987, -34.729]
  Call Extruder(206.22057)
  MoveL 3557 to (238.4, 42.45, 59.84) mm, rotated rx 180 ry 0 rz 180 deg; joints [-155.996, -76.194, -44.148, 41.397, 37.964, -34.799]
  MoveL 3558 to (238.4, 42.45, 59.84) mm, rotated rx 180 ry 0 rz 180 deg; joints [-155.996, -76.194, -44.148, 41.397, 37.964, -34.799]
  Call Extruder(206.42751)
  MoveL 3559 to (238.57, 42.75, 59.84) mm, rotated rx -180 ry 0 rz 180 deg; joints [-155.976, -76.233, -44.063, 41.463, 37.942, -34.87]
  MoveL 3560 to (238.57, 42.75, 59.84) mm, rotated rx -180 ry 0 rz 180 deg; joints [-155.976, -76.233, -44.063, 41.463, 37.942, -34.87]
  Call Extruder(206.63368)
  MoveL 3561 to (238.75, 43.06, 59.84) mm, rotated rx 180 ry 0 rz -180 deg; joints [-155.956, -76.272, -43.978, 41.529, 37.919, -34.94]
  MoveL 3562 to (238.75, 43.06, 59.84) mm, rotated rx 180 ry 0 rz -180 deg; joints [-155.956, -76.272, -43.978, 41.529, 37.919, -34.94]
  Call Extruder(206.81537)
  MoveL 3563 to (238.89, 43.33, 59.84) mm, rotated rx 180 ry 0 rz 180 deg; joints [-155.937, -76.306, -43.906, 41.588, 37.901, -35.002]
  MoveL 3564 to (238.89, 43.33, 59.84) mm, rotated rx 180 ry 0 rz 180 deg; joints [-155.937, -76.306, -43.906, 41.588, 37.901, -35.002]
  Call Extruder(206.97338)
  MoveL 3565 to (239, 43.58, 59.84) mm, rotated rx 180 ry 0 rz -180 deg; joints [-155.919, -76.333, -43.846, 41.639, 37.887, -35.056]
  MoveL 3566 to (239, 43.58, 59.84) mm, rotated rx 180 ry 0 rz -180 deg; joints [-155.919, -76.333, -43.846, 41.639, 37.887, -35.056]
  Call Extruder(207.13078)
  MoveL 3567 to (239.1, 43.83, 59.84) mm, rotated rx 180 ry 0 rz -180 deg; joints [-155.901, -76.361, -43.786, 41.69, 37.874, -35.11]
  MoveL 3568 to (239.1, 43.83, 59.84) mm, rotated rx 180 ry 0 rz -180 deg; joints [-155.901, -76.361, -43.786, 41.69, 37.874, -35.11]
  Call Extruder(207.31350)
  MoveL 3569 to (239.23, 44.12, 59.84) mm, rotated rx 180 ry 0 rz 180 deg; joints [-155.879, -76.393, -43.717, 41.75, 37.858, -35.172]
  MoveL 3570 to (239.23, 44.12, 59.84) mm, rotated rx 180 ry 0 rz 180 deg; joints [-155.879, -76.393, -43.717, 41.75, 37.858, -35.172]
  Call Extruder(207.49546)
  MoveL 3571 to (239.35, 44.42, 59.84) mm, rotated rx 180 ry 0 rz -180 deg; joints [-155.858, -76.425, -43.648, 41.811, 37.843, -35.235]
  MoveL 3572 to (239.35, 44.42, 59.84) mm, rotated rx 180 ry 0 rz -180 deg; joints [-155.858, -76.425, -43.648, 41.811, 37.843, -35.235]
  Call Extruder(207.64279)
  MoveL 3573 to (239.44, 44.66, 59.84) mm, rotated rx 180 ry 0 rz -180 deg; joints [-155.84, -76.45, -43.594, 41.859, 37.831, -35.285]
  MoveL 3574 to (239.44, 44.66, 59.84) mm, rotated rx 180 ry 0 rz -180 deg; joints [-155.84, -76.45, -43.594, 41.859, 37.831, -35.285]
  Call Extruder(207.75602)
  MoveL 3575 to (239.5, 44.85, 59.84) mm, rotated rx 180 ry 0 rz 180 deg; joints [-155.826, -76.468, -43.554, 41.897, 37.823, -35.324]
  MoveL 3576 to (239.5, 44.85, 59.84) mm, rotated rx 180 ry 0 rz 180 deg; joints [-155.826, -76.468, -43.554, 41.897, 37.823, -35.324]
  Call Extruder(207.86881)
  MoveL 3577 to (239.56, 45.03, 59.84) mm, rotated rx 180 ry 0 rz 180 deg; joints [-155.811, -76.487, -43.514, 41.935, 37.816, -35.363]
  MoveL 3578 to (239.56, 45.03, 59.84) mm, rotated rx 180 ry 0 rz 180 deg; joints [-155.811, -76.487, -43.514, 41.935, 37.816, -35.363]
  Call Extruder(207.98116)
  MoveL 3579 to (239.62, 45.22, 59.84) mm, rotated rx -180 ry 0 rz -180 deg; joints [-155.797, -76.505, -43.473, 41.972, 37.808, -35.401]
  MoveL 3580 to (239.62, 45.22, 59.84) mm, rotated rx -180 ry 0 rz -180 deg; joints [-155.797, -76.505, -43.473, 41.972, 37.808, -35.401]
  Call Extruder(208.09306)
  MoveL 3581 to (239.68, 45.41, 59.84) mm, rotated rx -180 ry 0 rz 180 deg; joints [-155.783, -76.524, -43.433, 42.01, 37.8, -35.44]
  MoveL 3582 to (239.68, 45.41, 59.84) mm, rotated rx -180 ry 0 rz 180 deg; joints [-155.783, -76.524, -43.433, 42.01, 37.8, -35.44]
  Call Extruder(208.21446)
  MoveL 3583 to (239.75, 45.62, 59.84) mm, rotated rx 180 ry 0 rz 180 deg; joints [-155.767, -76.544, -43.39, 42.051, 37.792, -35.482]
  MoveL 3584 to (239.75, 45.62, 59.84) mm, rotated rx 180 ry 0 rz 180 deg; joints [-155.767, -76.544, -43.39, 42.051, 37.792, -35.482]
  Call Extruder(208.34525)
  MoveL 3585 to (239.82, 45.84, 59.84) mm, rotated rx 180 ry 0 rz 180 deg; joints [-155.75, -76.566, -43.343, 42.096, 37.784, -35.527]
  MoveL 3586 to (239.82, 45.84, 59.84) mm, rotated rx 180 ry 0 rz 180 deg; joints [-155.75, -76.566, -43.343, 42.096, 37.784, -35.527]
  Call Extruder(208.47548)
  MoveL 3587 to (239.88, 46.06, 59.84) mm, rotated rx 180 ry 0 rz 180 deg; joints [-155.733, -76.587, -43.297, 42.14, 37.775, -35.572]
  MoveL 3588 to (239.88, 46.06, 59.84) mm, rotated rx 180 ry 0 rz 180 deg; joints [-155.733, -76.587, -43.297, 42.14, 37.775, -35.572]
  Call Extruder(208.60514)
  MoveL 3589 to (239.95, 46.29, 59.84) mm, rotated rx -180 ry 0 rz 180 deg; joints [-155.715, -76.609, -43.251, 42.184, 37.767, -35.618]
  MoveL 3590 to (239.95, 46.29, 59.84) mm, rotated rx -180 ry 0 rz 180 deg; joints [-155.715, -76.609, -43.251, 42.184, 37.767, -35.618]
  Call Extruder(208.73424)
  MoveL 3591 to (240.02, 46.51, 59.84) mm, rotated rx 180 ry 0 rz 180 deg; joints [-155.698, -76.63, -43.204, 42.229, 37.758, -35.663]
  MoveL 3592 to (240.02, 46.51, 59.84) mm, rotated rx 180 ry 0 rz 180 deg; joints [-155.698, -76.63, -43.204, 42.229, 37.758, -35.663]
  Call Extruder(208.84929)
  MoveL 3593 to (240.06, 46.72, 59.84) mm, rotated rx -180 ry 0 rz -180 deg; joints [-155.682, -76.648, -43.166, 42.268, 37.753, -35.703]
  MoveL 3594 to (240.06, 46.72, 59.84) mm, rotated rx -180 ry 0 rz -180 deg; joints [-155.682, -76.648, -43.166, 42.268, 37.753, -35.703]
  Call Extruder(208.96389)
  MoveL 3595 to (240.11, 46.92, 59.84) mm, rotated rx -180 ry 0 rz 180 deg; joints [-155.665, -76.665, -43.129, 42.308, 37.747, -35.742]
  MoveL 3596 to (240.11, 46.92, 59.84) mm, rotated rx -180 ry 0 rz 180 deg; joints [-155.665, -76.665, -43.129, 42.308, 37.747, -35.742]
  Call Extruder(209.07804)
  MoveL 3597 to (240.15, 47.12, 59.84) mm, rotated rx 180 ry 0 rz 180 deg; joints [-155.649, -76.683, -43.091, 42.347, 37.742, -35.782]
  MoveL 3598 to (240.15, 47.12, 59.84) mm, rotated rx 180 ry 0 rz 180 deg; joints [-155.649, -76.683, -43.091, 42.347, 37.742, -35.782]
  Call Extruder(209.19174)
  MoveL 3599 to (240.2, 47.33, 59.84) mm, rotated rx -180 ry 0 rz 180 deg; joints [-155.633, -76.7, -43.053, 42.386, 37.736, -35.821]
  MoveL 3600 to (240.2, 47.33, 59.84) mm, rotated rx -180 ry 0 rz 180 deg; joints [-155.633, -76.7, -43.053, 42.386, 37.736, -35.821]
  Call Extruder(209.31715)
  MoveL 3601 to (240.24, 47.55, 59.84) mm, rotated rx 180 ry 0 rz 180 deg; joints [-155.614, -76.72, -43.011, 42.43, 37.731, -35.865]
  MoveL 3602 to (240.24, 47.55, 59.84) mm, rotated rx 180 ry 0 rz 180 deg; joints [-155.614, -76.72, -43.011, 42.43, 37.731, -35.865]
  Call Extruder(209.45413)
  MoveL 3603 to (240.29, 47.8, 59.84) mm, rotated rx 180 ry 0 rz 180 deg; joints [-155.594, -76.74, -42.966, 42.478, 37.725, -35.912]
  MoveL 3604 to (240.29, 47.8, 59.84) mm, rotated rx 180 ry 0 rz 180 deg; joints [-155.594, -76.74, -42.966, 42.478, 37.725, -35.912]
  Call Extruder(209.59050)
  MoveL 3605 to (240.34, 48.05, 59.84) mm, rotated rx 180 ry 0 rz 180 deg; joints [-155.574, -76.761, -42.921, 42.525, 37.719, -35.96]
  MoveL 3606 to (240.34, 48.05, 59.84) mm, rotated rx 180 ry 0 rz 180 deg; joints [-155.574, -76.761, -42.921, 42.525, 37.719, -35.96]
  Call Extruder(209.72625)
  MoveL 3607 to (240.39, 48.3, 59.84) mm, rotated rx 180 ry 0 rz 180 deg; joints [-155.554, -76.782, -42.876, 42.573, 37.713, -36.008]
  MoveL 3608 to (240.39, 48.3, 59.84) mm, rotated rx 180 ry 0 rz 180 deg; joints [-155.554, -76.782, -42.876, 42.573, 37.713, -36.008]
  Call Extruder(209.86140)
  MoveL 3609 to (240.44, 48.55, 59.84) mm, rotated rx -180 ry 0 rz 180 deg; joints [-155.534, -76.803, -42.831, 42.621, 37.707, -36.056]
  MoveL 3610 to (240.44, 48.55, 59.84) mm, rotated rx -180 ry 0 rz 180 deg; joints [-155.534, -76.803, -42.831, 42.621, 37.707, -36.056]
  Call Extruder(209.99594)
  MoveL 3611 to (240.49, 48.8, 59.84) mm, rotated rx -180 ry 0 rz -180 deg; joints [-155.514, -76.824, -42.786, 42.669, 37.701, -36.104]
  MoveL 3612 to (240.49, 48.8, 59.84) mm, rotated rx -180 ry 0 rz -180 deg; joints [-155.514, -76.824, -42.786, 42.669, 37.701, -36.104]
  Call Extruder(210.12986)
  MoveL 3613 to (240.54, 49.05, 59.84) mm, rotated rx -180 ry 0 rz 180 deg; joints [-155.494, -76.845, -42.741, 42.716, 37.695, -36.152]
  MoveL 3614 to (240.54, 49.05, 59.84) mm, rotated rx -180 ry 0 rz 180 deg; joints [-155.494, -76.845, -42.741, 42.716, 37.695, -36.152]
  Call Extruder(210.27773)
  MoveL 3615 to (240.59, 49.33, 59.84) mm, rotated rx 180 ry 0 rz 180 deg; joints [-155.471, -76.868, -42.692, 42.769, 37.689, -36.204]
  MoveL 3616 to (240.59, 49.33, 59.84) mm, rotated rx 180 ry 0 rz 180 deg; joints [-155.471, -76.868, -42.692, 42.769, 37.689, -36.204]
  Call Extruder(210.43947)
  MoveL 3617 to (240.64, 49.63, 59.84) mm, rotated rx 180 ry 0 rz -180 deg; joints [-155.446, -76.892, -42.639, 42.827, 37.683, -36.262]
  MoveL 3618 to (240.64, 49.63, 59.84) mm, rotated rx 180 ry 0 rz -180 deg; joints [-155.446, -76.892, -42.639, 42.827, 37.683, -36.262]
  Call Extruder(210.60049)
  MoveL 3619 to (240.69, 49.94, 59.84) mm, rotated rx -180 ry 0 rz 180 deg; joints [-155.421, -76.916, -42.587, 42.885, 37.677, -36.319]
  MoveL 3620 to (240.69, 49.94, 59.84) mm, rotated rx -180 ry 0 rz 180 deg; joints [-155.421, -76.916, -42.587, 42.885, 37.677, -36.319]
  Call Extruder(210.76078)
  MoveL 3621 to (240.74, 50.24, 59.84) mm, rotated rx 180 ry 0 rz 180 deg; joints [-155.396, -76.941, -42.535, 42.943, 37.672, -36.376]
  MoveL 3622 to (240.74, 50.24, 59.84) mm, rotated rx 180 ry 0 rz 180 deg; joints [-155.396, -76.941, -42.535, 42.943, 37.672, -36.376]
  Call Extruder(210.92034)
  MoveL 3623 to (240.78, 50.55, 59.84) mm, rotated rx 180 ry 0 rz 180 deg; joints [-155.371, -76.965, -42.482, 43.001, 37.666, -36.434]
  MoveL 3624 to (240.78, 50.55, 59.84) mm, rotated rx 180 ry 0 rz 180 deg; joints [-155.371, -76.965, -42.482, 43.001, 37.666, -36.434]
  Call Extruder(211.07917)
  MoveL 3625 to (240.83, 50.86, 59.84) mm, rotated rx -180 ry 0 rz 180 deg; joints [-155.346, -76.99, -42.429, 43.059, 37.66, -36.492]
  MoveL 3626 to (240.83, 50.86, 59.84) mm, rotated rx -180 ry 0 rz 180 deg; joints [-155.346, -76.99, -42.429, 43.059, 37.66, -36.492]
  Call Extruder(211.25784)
  MoveL 3627 to (240.88, 51.2, 59.84) mm, rotated rx -180 ry 0 rz 180 deg; joints [-155.317, -77.016, -42.372, 43.123, 37.655, -36.556]
  MoveL 3628 to (240.88, 51.2, 59.84) mm, rotated rx -180 ry 0 rz 180 deg; joints [-155.317, -77.016, -42.372, 43.123, 37.655, -36.556]
  Call Extruder(211.45628)
  MoveL 3629 to (240.93, 51.59, 59.84) mm, rotated rx 180 ry 0 rz -180 deg; joints [-155.285, -77.045, -42.309, 43.196, 37.65, -36.627]
  MoveL 3630 to (240.93, 51.59, 59.84) mm, rotated rx 180 ry 0 rz -180 deg; joints [-155.285, -77.045, -42.309, 43.196, 37.65, -36.627]
  Call Extruder(211.65386)
  MoveL 3631 to (240.97, 51.98, 59.84) mm, rotated rx 180 ry 0 rz -180 deg; joints [-155.252, -77.075, -42.246, 43.268, 37.645, -36.698]
  MoveL 3632 to (240.97, 51.98, 59.84) mm, rotated rx 180 ry 0 rz -180 deg; joints [-155.252, -77.075, -42.246, 43.268, 37.645, -36.698]
  Call Extruder(211.85056)
  MoveL 3633 to (241.02, 52.36, 59.84) mm, rotated rx -180 ry 0 rz 180 deg; joints [-155.22, -77.104, -42.184, 43.34, 37.639, -36.77]
  MoveL 3634 to (241.02, 52.36, 59.84) mm, rotated rx -180 ry 0 rz 180 deg; joints [-155.22, -77.104, -42.184, 43.34, 37.639, -36.77]
  Call Extruder(212.04640)
  MoveL 3635 to (241.06, 52.75, 59.84) mm, rotated rx 180 ry 0 rz 180 deg; joints [-155.188, -77.133, -42.121, 43.413, 37.634, -36.841]
  MoveL 3636 to (241.06, 52.75, 59.84) mm, rotated rx 180 ry 0 rz 180 deg; joints [-155.188, -77.133, -42.121, 43.413, 37.634, -36.841]
  Call Extruder(212.34184)
  MoveL 3637 to (241.11, 53.34, 59.84) mm, rotated rx 180 ry 0 rz 180 deg; joints [-155.138, -77.175, -42.031, 43.521, 37.63, -36.947]
  MoveL 3638 to (241.11, 53.34, 59.84) mm, rotated rx 180 ry 0 rz 180 deg; joints [-155.138, -77.175, -42.031, 43.521, 37.63, -36.947]
  Call Extruder(212.63595)
  MoveL 3639 to (241.16, 53.93, 59.84) mm, rotated rx 180 ry 0 rz 180 deg; joints [-155.088, -77.216, -41.942, 43.629, 37.625, -37.053]
  MoveL 3640 to (241.16, 53.93, 59.84) mm, rotated rx 180 ry 0 rz 180 deg; joints [-155.088, -77.216, -41.942, 43.629, 37.625, -37.053]
  Call Extruder(212.92873)
  MoveL 3641 to (241.2, 54.52, 59.84) mm, rotated rx 180 ry 0 rz -180 deg; joints [-155.038, -77.258, -41.851, 43.738, 37.62, -37.159]
  MoveL 3642 to (241.2, 54.52, 59.84) mm, rotated rx 180 ry 0 rz -180 deg; joints [-155.038, -77.258, -41.851, 43.738, 37.62, -37.159]
  Call Extruder(213.50218)
  MoveL 3643 to (241.25, 55.68, 59.84) mm, rotated rx -180 ry 0 rz 180 deg; joints [-154.938, -77.335, -41.686, 43.948, 37.617, -37.363]
  MoveL 3644 to (241.25, 55.68, 59.84) mm, rotated rx -180 ry 0 rz 180 deg; joints [-154.938, -77.335, -41.686, 43.948, 37.617, -37.363]
  Call Extruder(214.21601)
  MoveL 3645 to (241.29, 57.14, 59.84) mm, rotated rx 180 ry 0 rz 180 deg; joints [-154.812, -77.43, -41.482, 44.209, 37.616, -37.616]
  Call Extruder(256.28089)
  MoveL 3646 to (241.29, 142.86, 59.84) mm, rotated rx -180 ry 0 rz 180 deg; joints [-147.778, -84.499, -26.665, 60.195, 37.914, -54.017]
  Call Extruder(256.70932)
  MoveL 3647 to (241.27, 143.73, 59.84) mm, rotated rx 180 ry 0 rz 180 deg; joints [-147.711, -84.592, -26.473, 60.369, 37.92, -54.207]
  MoveL 3648 to (241.27, 143.73, 59.84) mm, rotated rx 180 ry 0 rz 180 deg; joints [-147.711, -84.592, -26.473, 60.369, 37.92, -54.207]
  Call Extruder(257.28277)
  MoveL 3649 to (241.22, 144.9, 59.84) mm, rotated rx -180 ry 0 rz 180 deg; joints [-147.62, -84.714, -26.223, 60.598, 37.931, -54.456]
  MoveL 3650 to (241.22, 144.9, 59.84) mm, rotated rx -180 ry 0 rz 180 deg; joints [-147.62, -84.714, -26.223, 60.598, 37.931, -54.456]
  Call Extruder(257.71711)
  MoveL 3651 to (241.18, 145.77, 59.84) mm, rotated rx 180 ry 0 rz 180 deg; joints [-147.551, -84.804, -26.038, 60.769, 37.941, -54.642]
  MoveL 3652 to (241.18, 145.77, 59.84) mm, rotated rx 180 ry 0 rz 180 deg; joints [-147.551, -84.804, -26.038, 60.769, 37.941, -54.642]
  Call Extruder(258.01122)
  MoveL 3653 to (241.13, 146.36, 59.84) mm, rotated rx 180 ry 0 rz -180 deg; joints [-147.504, -84.863, -25.919, 60.882, 37.95, -54.764]
  MoveL 3654 to (241.13, 146.36, 59.84) mm, rotated rx 180 ry 0 rz -180 deg; joints [-147.504, -84.863, -25.919, 60.882, 37.95, -54.764]
  Call Extruder(258.30666)
  MoveL 3655 to (241.09, 146.95, 59.84) mm, rotated rx -180 ry 0 rz -180 deg; joints [-147.457, -84.921, -25.798, 60.995, 37.958, -54.886]
  MoveL 3656 to (241.09, 146.95, 59.84) mm, rotated rx -180 ry 0 rz -180 deg; joints [-147.457, -84.921, -25.798, 60.995, 37.958, -54.886]
  Call Extruder(258.55291)
  MoveL 3657 to (241.04, 147.44, 59.84) mm, rotated rx 180 ry 0 rz 180 deg; joints [-147.417, -84.969, -25.701, 61.088, 37.966, -54.986]
  MoveL 3658 to (241.04, 147.44, 59.84) mm, rotated rx 180 ry 0 rz 180 deg; joints [-147.417, -84.969, -25.701, 61.088, 37.966, -54.986]
  Call Extruder(258.74962)
  MoveL 3659 to (240.99, 147.83, 59.84) mm, rotated rx -180 ry 0 rz 180 deg; joints [-147.386, -85.005, -25.627, 61.16, 37.974, -55.063]
  MoveL 3660 to (240.99, 147.83, 59.84) mm, rotated rx -180 ry 0 rz 180 deg; joints [-147.386, -85.005, -25.627, 61.16, 37.974, -55.063]
  Call Extruder(258.94719)
  MoveL 3661 to (240.95, 148.22, 59.84) mm, rotated rx 180 ry 0 rz 180 deg; joints [-147.354, -85.041, -25.553, 61.231, 37.981, -55.14]
  MoveL 3662 to (240.95, 148.22, 59.84) mm, rotated rx 180 ry 0 rz 180 deg; joints [-147.354, -85.041, -25.553, 61.231, 37.981, -55.14]
  Call Extruder(259.14563)
  MoveL 3663 to (240.9, 148.6, 59.84) mm, rotated rx 180 ry 0 rz -180 deg; joints [-147.322, -85.078, -25.479, 61.304, 37.989, -55.218]
  MoveL 3664 to (240.9, 148.6, 59.84) mm, rotated rx 180 ry 0 rz -180 deg; joints [-147.322, -85.078, -25.479, 61.304, 37.989, -55.218]
  Call Extruder(259.34494)
  MoveL 3665 to (240.86, 148.99, 59.84) mm, rotated rx -180 ry 0 rz 180 deg; joints [-147.291, -85.114, -25.404, 61.376, 37.997, -55.295]
  MoveL 3666 to (240.86, 148.99, 59.84) mm, rotated rx -180 ry 0 rz 180 deg; joints [-147.291, -85.114, -25.404, 61.376, 37.997, -55.295]
  Call Extruder(259.50377)
  MoveL 3667 to (240.81, 149.3, 59.84) mm, rotated rx -180 ry 0 rz 180 deg; joints [-147.265, -85.141, -25.349, 61.431, 38.004, -55.354]
  MoveL 3668 to (240.81, 149.3, 59.84) mm, rotated rx -180 ry 0 rz 180 deg; joints [-147.265, -85.141, -25.349, 61.431, 38.004, -55.354]
  Call Extruder(259.66333)
  MoveL 3669 to (240.76, 149.6, 59.84) mm, rotated rx 180 ry 0 rz 180 deg; joints [-147.24, -85.167, -25.295, 61.486, 38.012, -55.412]
  MoveL 3670 to (240.76, 149.6, 59.84) mm, rotated rx 180 ry 0 rz 180 deg; joints [-147.24, -85.167, -25.295, 61.486, 38.012, -55.412]
  Call Extruder(259.82362)
  MoveL 3671 to (240.71, 149.91, 59.84) mm, rotated rx 180 ry 0 rz 180 deg; joints [-147.214, -85.194, -25.24, 61.54, 38.02, -55.47]
  MoveL 3672 to (240.71, 149.91, 59.84) mm, rotated rx 180 ry 0 rz 180 deg; joints [-147.214, -85.194, -25.24, 61.54, 38.02, -55.47]
  Call Extruder(259.98464)
  MoveL 3673 to (240.66, 150.21, 59.84) mm, rotated rx -180 ry 0 rz 180 deg; joints [-147.189, -85.221, -25.185, 61.595, 38.027, -55.529]
  MoveL 3674 to (240.66, 150.21, 59.84) mm, rotated rx -180 ry 0 rz 180 deg; joints [-147.189, -85.221, -25.185, 61.595, 38.027, -55.529]
  Call Extruder(260.14638)
  MoveL 3675 to (240.61, 150.52, 59.84) mm, rotated rx -180 ry 0 rz 180 deg; joints [-147.163, -85.248, -25.13, 61.651, 38.035, -55.588]
  MoveL 3676 to (240.61, 150.52, 59.84) mm, rotated rx -180 ry 0 rz 180 deg; joints [-147.163, -85.248, -25.13, 61.651, 38.035, -55.588]
  Call Extruder(260.30885)
  MoveL 3677 to (240.56, 150.83, 59.84) mm, rotated rx -180 ry 0 rz -180 deg; joints [-147.138, -85.275, -25.075, 61.706, 38.043, -55.646]
  MoveL 3678 to (240.56, 150.83, 59.84) mm, rotated rx -180 ry 0 rz -180 deg; joints [-147.138, -85.275, -25.075, 61.706, 38.043, -55.646]
  Call Extruder(260.44278)
  MoveL 3679 to (240.52, 151.07, 59.84) mm, rotated rx 180 ry 0 rz 180 deg; joints [-147.117, -85.295, -25.033, 61.749, 38.05, -55.692]
  MoveL 3680 to (240.52, 151.07, 59.84) mm, rotated rx 180 ry 0 rz 180 deg; joints [-147.117, -85.295, -25.033, 61.749, 38.05, -55.692]
  Call Extruder(260.57732)
  MoveL 3681 to (240.47, 151.32, 59.84) mm, rotated rx -180 ry 0 rz 180 deg; joints [-147.095, -85.316, -24.992, 61.792, 38.058, -55.737]
  MoveL 3682 to (240.47, 151.32, 59.84) mm, rotated rx -180 ry 0 rz 180 deg; joints [-147.095, -85.316, -24.992, 61.792, 38.058, -55.737]
  Call Extruder(260.71246)
  MoveL 3683 to (240.42, 151.57, 59.84) mm, rotated rx -180 ry 0 rz 180 deg; joints [-147.074, -85.336, -24.951, 61.835, 38.065, -55.783]
  MoveL 3684 to (240.42, 151.57, 59.84) mm, rotated rx -180 ry 0 rz 180 deg; joints [-147.074, -85.336, -24.951, 61.835, 38.065, -55.783]
  Call Extruder(260.84822)
  MoveL 3685 to (240.37, 151.82, 59.84) mm, rotated rx 180 ry 0 rz -180 deg; joints [-147.053, -85.356, -24.909, 61.878, 38.073, -55.828]
  MoveL 3686 to (240.37, 151.82, 59.84) mm, rotated rx 180 ry 0 rz -180 deg; joints [-147.053, -85.356, -24.909, 61.878, 38.073, -55.828]
  Call Extruder(260.98459)
  MoveL 3687 to (240.32, 152.07, 59.84) mm, rotated rx -180 ry 0 rz -180 deg; joints [-147.032, -85.377, -24.867, 61.922, 38.08, -55.874]
  MoveL 3688 to (240.32, 152.07, 59.84) mm, rotated rx -180 ry 0 rz -180 deg; joints [-147.032, -85.377, -24.867, 61.922, 38.08, -55.874]
  Call Extruder(261.12157)
  MoveL 3689 to (240.27, 152.32, 59.84) mm, rotated rx 180 ry 0 rz -180 deg; joints [-147.011, -85.397, -24.825, 61.965, 38.088, -55.92]
  MoveL 3690 to (240.27, 152.32, 59.84) mm, rotated rx 180 ry 0 rz -180 deg; joints [-147.011, -85.397, -24.825, 61.965, 38.088, -55.92]
  Call Extruder(261.25915)
  MoveL 3691 to (240.22, 152.57, 59.84) mm, rotated rx 180 ry 0 rz 180 deg; joints [-146.989, -85.418, -24.784, 62.008, 38.095, -55.965]
  MoveL 3692 to (240.22, 152.57, 59.84) mm, rotated rx 180 ry 0 rz 180 deg; joints [-146.989, -85.418, -24.784, 62.008, 38.095, -55.965]
  Call Extruder(261.37285)
  MoveL 3693 to (240.17, 152.77, 59.84) mm, rotated rx -180 ry 0 rz 180 deg; joints [-146.972, -85.434, -24.75, 62.043, 38.102, -56.002]
  MoveL 3694 to (240.17, 152.77, 59.84) mm, rotated rx -180 ry 0 rz 180 deg; joints [-146.972, -85.434, -24.75, 62.043, 38.102, -56.002]
  Call Extruder(261.48700)
  MoveL 3695 to (240.13, 152.98, 59.84) mm, rotated rx 180 ry 0 rz -180 deg; joints [-146.954, -85.45, -24.718, 62.078, 38.109, -56.038]
  MoveL 3696 to (240.13, 152.98, 59.84) mm, rotated rx 180 ry 0 rz -180 deg; joints [-146.954, -85.45, -24.718, 62.078, 38.109, -56.038]
  Call Extruder(261.60161)
  MoveL 3697 to (240.08, 153.18, 59.84) mm, rotated rx 180 ry 0 rz 180 deg; joints [-146.937, -85.466, -24.685, 62.113, 38.115, -56.075]
  MoveL 3698 to (240.08, 153.18, 59.84) mm, rotated rx 180 ry 0 rz 180 deg; joints [-146.937, -85.466, -24.685, 62.113, 38.115, -56.075]
  Call Extruder(261.71666)
  MoveL 3699 to (240.04, 153.39, 59.84) mm, rotated rx 180 ry 0 rz -180 deg; joints [-146.919, -85.482, -24.652, 62.148, 38.122, -56.112]
  MoveL 3700 to (240.04, 153.39, 59.84) mm, rotated rx 180 ry 0 rz -180 deg; joints [-146.919, -85.482, -24.652, 62.148, 38.122, -56.112]
  Call Extruder(261.83888)
  MoveL 3701 to (239.98, 153.6, 59.84) mm, rotated rx -180 ry 0 rz -180 deg; joints [-146.9, -85.497, -24.62, 62.183, 38.13, -56.148]
  MoveL 3702 to (239.98, 153.6, 59.84) mm, rotated rx -180 ry 0 rz -180 deg; joints [-146.9, -85.497, -24.62, 62.183, 38.13, -56.148]
  Call Extruder(261.96855)
  MoveL 3703 to (239.92, 153.82, 59.84) mm, rotated rx -180 ry 0 rz -180 deg; joints [-146.88, -85.512, -24.591, 62.218, 38.14, -56.183]
  MoveL 3704 to (239.92, 153.82, 59.84) mm, rotated rx -180 ry 0 rz -180 deg; joints [-146.88, -85.512, -24.591, 62.218, 38.14, -56.183]
  Call Extruder(262.09877)
  MoveL 3705 to (239.85, 154.05, 59.84) mm, rotated rx 180 ry 0 rz 180 deg; joints [-146.86, -85.526, -24.562, 62.252, 38.15, -56.219]
  MoveL 3706 to (239.85, 154.05, 59.84) mm, rotated rx 180 ry 0 rz 180 deg; joints [-146.86, -85.526, -24.562, 62.252, 38.15, -56.219]
  Call Extruder(262.22956)
  MoveL 3707 to (239.78, 154.27, 59.84) mm, rotated rx 180 ry 0 rz -180 deg; joints [-146.84, -85.541, -24.532, 62.288, 38.16, -56.255]
  MoveL 3708 to (239.78, 154.27, 59.84) mm, rotated rx 180 ry 0 rz -180 deg; joints [-146.84, -85.541, -24.532, 62.288, 38.16, -56.255]
  Call Extruder(262.36092)
  MoveL 3709 to (239.71, 154.5, 59.84) mm, rotated rx 180 ry 0 rz 180 deg; joints [-146.82, -85.555, -24.503, 62.323, 38.169, -56.291]
  MoveL 3710 to (239.71, 154.5, 59.84) mm, rotated rx 180 ry 0 rz 180 deg; joints [-146.82, -85.555, -24.503, 62.323, 38.169, -56.291]
  Call Extruder(262.47282)
  MoveL 3711 to (239.65, 154.68, 59.84) mm, rotated rx -180 ry 0 rz 180 deg; joints [-146.803, -85.566, -24.48, 62.351, 38.178, -56.32]
  MoveL 3712 to (239.65, 154.68, 59.84) mm, rotated rx -180 ry 0 rz 180 deg; joints [-146.803, -85.566, -24.48, 62.351, 38.178, -56.32]
  Call Extruder(262.58516)
  MoveL 3713 to (239.59, 154.87, 59.84) mm, rotated rx 180 ry 0 rz 180 deg; joints [-146.785, -85.578, -24.456, 62.38, 38.187, -56.349]
  MoveL 3714 to (239.59, 154.87, 59.84) mm, rotated rx 180 ry 0 rz 180 deg; joints [-146.785, -85.578, -24.456, 62.38, 38.187, -56.349]
  Call Extruder(262.69795)
  MoveL 3715 to (239.53, 155.06, 59.84) mm, rotated rx 180 ry 0 rz -180 deg; joints [-146.768, -85.589, -24.433, 62.409, 38.196, -56.378]
  MoveL 3716 to (239.53, 155.06, 59.84) mm, rotated rx 180 ry 0 rz -180 deg; joints [-146.768, -85.589, -24.433, 62.409, 38.196, -56.378]
  Call Extruder(262.81119)
  MoveL 3717 to (239.47, 155.25, 59.84) mm, rotated rx -180 ry 0 rz 180 deg; joints [-146.751, -85.601, -24.41, 62.438, 38.204, -56.407]
  MoveL 3718 to (239.47, 155.25, 59.84) mm, rotated rx -180 ry 0 rz 180 deg; joints [-146.751, -85.601, -24.41, 62.438, 38.204, -56.407]
  Call Extruder(262.92487)
  MoveL 3719 to (239.41, 155.44, 59.84) mm, rotated rx 180 ry 0 rz 180 deg; joints [-146.734, -85.612, -24.386, 62.467, 38.213, -56.436]
  MoveL 3720 to (239.41, 155.44, 59.84) mm, rotated rx 180 ry 0 rz 180 deg; joints [-146.734, -85.612, -24.386, 62.467, 38.213, -56.436]
  Call Extruder(263.10683)
  MoveL 3721 to (239.29, 155.73, 59.84) mm, rotated rx -180 ry 0 rz 180 deg; joints [-146.706, -85.625, -24.36, 62.507, 38.23, -56.475]
  MoveL 3722 to (239.29, 155.73, 59.84) mm, rotated rx -180 ry 0 rz 180 deg; joints [-146.706, -85.625, -24.36, 62.507, 38.23, -56.475]
  Call Extruder(263.28954)
  MoveL 3723 to (239.17, 156.02, 59.84) mm, rotated rx 180 ry 0 rz -180 deg; joints [-146.678, -85.638, -24.333, 62.547, 38.247, -56.514]
  MoveL 3724 to (239.17, 156.02, 59.84) mm, rotated rx 180 ry 0 rz -180 deg; joints [-146.678, -85.638, -24.333, 62.547, 38.247, -56.514]
  Call Extruder(263.45997)
  MoveL 3725 to (239.05, 156.29, 59.84) mm, rotated rx 180 ry 0 rz 180 deg; joints [-146.652, -85.65, -24.309, 62.584, 38.263, -56.55]
  MoveL 3726 to (239.05, 156.29, 59.84) mm, rotated rx 180 ry 0 rz 180 deg; joints [-146.652, -85.65, -24.309, 62.584, 38.263, -56.55]
  Call Extruder(263.61798)
  MoveL 3727 to (238.94, 156.54, 59.84) mm, rotated rx 180 ry 0 rz 180 deg; joints [-146.628, -85.661, -24.288, 62.617, 38.278, -56.582]
  MoveL 3728 to (238.94, 156.54, 59.84) mm, rotated rx 180 ry 0 rz 180 deg; joints [-146.628, -85.661, -24.288, 62.617, 38.278, -56.582]
  Call Extruder(263.77659)
  MoveL 3729 to (238.84, 156.79, 59.84) mm, rotated rx 180 ry 0 rz 180 deg; joints [-146.604, -85.671, -24.266, 62.651, 38.293, -56.615]
  MoveL 3730 to (238.84, 156.79, 59.84) mm, rotated rx 180 ry 0 rz 180 deg; joints [-146.604, -85.671, -24.266, 62.651, 38.293, -56.615]
  Call Extruder(263.98276)
  MoveL 3731 to (238.66, 157.09, 59.84) mm, rotated rx 180 ry 0 rz 180 deg; joints [-146.573, -85.676, -24.256, 62.684, 38.317, -56.644]
  MoveL 3732 to (238.66, 157.09, 59.84) mm, rotated rx 180 ry 0 rz 180 deg; joints [-146.573, -85.676, -24.256, 62.684, 38.317, -56.644]
  Call Extruder(264.18971)
  MoveL 3733 to (238.49, 157.4, 59.84) mm, rotated rx 180 ry 0 rz 180 deg; joints [-146.542, -85.68, -24.247, 62.718, 38.341, -56.672]
  MoveL 3734 to (238.49, 157.4, 59.84) mm, rotated rx 180 ry 0 rz 180 deg; joints [-146.542, -85.68, -24.247, 62.718, 38.341, -56.672]
  Call Extruder(264.39743)
  MoveL 3735 to (238.31, 157.7, 59.84) mm, rotated rx 180 ry 0 rz -180 deg; joints [-146.51, -85.685, -24.237, 62.751, 38.365, -56.701]
  MoveL 3736 to (238.31, 157.7, 59.84) mm, rotated rx 180 ry 0 rz -180 deg; joints [-146.51, -85.685, -24.237, 62.751, 38.365, -56.701]
  Call Extruder(264.60594)
  MoveL 3737 to (238.14, 158.01, 59.84) mm, rotated rx 180 ry 0 rz 180 deg; joints [-146.479, -85.69, -24.228, 62.784, 38.389, -56.73]
  MoveL 3738 to (238.14, 158.01, 59.84) mm, rotated rx 180 ry 0 rz 180 deg; joints [-146.479, -85.69, -24.228, 62.784, 38.389, -56.73]
  Call Extruder(264.78548)
  MoveL 3739 to (237.96, 158.25, 59.84) mm, rotated rx 180 ry 0 rz 180 deg; joints [-146.452, -85.687, -24.233, 62.805, 38.413, -56.745]
  MoveL 3740 to (237.96, 158.25, 59.84) mm, rotated rx 180 ry 0 rz 180 deg; joints [-146.452, -85.687, -24.233, 62.805, 38.413, -56.745]
  Call Extruder(265.11889)
  MoveL 3741 to (237.63, 158.7, 59.84) mm, rotated rx -180 ry 0 rz 180 deg; joints [-146.402, -85.682, -24.244, 62.843, 38.457, -56.772]
  MoveL 3742 to (237.63, 158.7, 59.84) mm, rotated rx -180 ry 0 rz 180 deg; joints [-146.402, -85.682, -24.244, 62.843, 38.457, -56.772]
  Call Extruder(265.45348)
  MoveL 3743 to (237.3, 159.15, 59.84) mm, rotated rx -180 ry 0 rz -180 deg; joints [-146.352, -85.677, -24.254, 62.881, 38.501, -56.799]
  Call Extruder(266.28143)
  MoveL 3744 to (236.39, 160.19, 59.84) mm, rotated rx -180 ry 0 rz 180 deg; joints [-146.229, -85.637, -24.336, 62.942, 38.623, -56.823]
  Call Extruder(267.10937)
  MoveL 3745 to (235.35, 161.1, 59.84) mm, rotated rx -180 ry 0 rz 180 deg; joints [-146.109, -85.559, -24.495, 62.957, 38.76, -56.789]
  Call Extruder(267.27668)
  MoveL 3746 to (235.13, 161.27, 59.84) mm, rotated rx 180 ry 0 rz 180 deg; joints [-146.086, -85.538, -24.538, 62.953, 38.79, -56.774]
  MoveL 3747 to (235.13, 161.27, 59.84) mm, rotated rx 180 ry 0 rz 180 deg; joints [-146.086, -85.538, -24.538, 62.953, 38.79, -56.774]
  Call Extruder(267.61010)
  MoveL 3748 to (234.68, 161.59, 59.84) mm, rotated rx -180 ry 0 rz 180 deg; joints [-146.039, -85.496, -24.624, 62.946, 38.849, -56.744]
  MoveL 3749 to (234.68, 161.59, 59.84) mm, rotated rx -180 ry 0 rz 180 deg; joints [-146.039, -85.496, -24.624, 62.946, 38.849, -56.744]
  Call Extruder(267.94234)
  MoveL 3750 to (234.22, 161.92, 59.84) mm, rotated rx 180 ry 0 rz 180 deg; joints [-145.992, -85.454, -24.709, 62.939, 38.908, -56.715]
  MoveL 3751 to (234.22, 161.92, 59.84) mm, rotated rx 180 ry 0 rz 180 deg; joints [-145.992, -85.454, -24.709, 62.939, 38.908, -56.715]
  Call Extruder(268.06000)
  MoveL 3752 to (234.05, 162.02, 59.84) mm, rotated rx -180 ry 0 rz 180 deg; joints [-145.976, -85.435, -24.747, 62.931, 38.93, -56.698]
  MoveL 3753 to (234.05, 162.02, 59.84) mm, rotated rx -180 ry 0 rz 180 deg; joints [-145.976, -85.435, -24.747, 62.931, 38.93, -56.698]
  Call Extruder(268.26773)
  MoveL 3754 to (233.75, 162.2, 59.84) mm, rotated rx -180 ry 0 rz 180 deg; joints [-145.947, -85.402, -24.816, 62.918, 38.97, -56.668]
  MoveL 3755 to (233.75, 162.2, 59.84) mm, rotated rx -180 ry 0 rz 180 deg; joints [-145.947, -85.402, -24.816, 62.918, 38.97, -56.668]
  Call Extruder(268.47467)
  MoveL 3756 to (233.45, 162.37, 59.84) mm, rotated rx 180 ry 0 rz -180 deg; joints [-145.919, -85.368, -24.884, 62.904, 39.01, -56.637]
  MoveL 3757 to (233.45, 162.37, 59.84) mm, rotated rx 180 ry 0 rz -180 deg; joints [-145.919, -85.368, -24.884, 62.904, 39.01, -56.637]
  Call Extruder(268.68084)
  MoveL 3758 to (233.14, 162.55, 59.84) mm, rotated rx -180 ry 0 rz -180 deg; joints [-145.891, -85.335, -24.952, 62.891, 39.049, -56.608]
  MoveL 3759 to (233.14, 162.55, 59.84) mm, rotated rx -180 ry 0 rz -180 deg; joints [-145.891, -85.335, -24.952, 62.891, 39.049, -56.608]
  Call Extruder(268.86251)
  MoveL 3760 to (232.87, 162.69, 59.84) mm, rotated rx 180 ry 0 rz 180 deg; joints [-145.866, -85.303, -25.018, 62.875, 39.085, -56.576]
  MoveL 3761 to (232.87, 162.69, 59.84) mm, rotated rx 180 ry 0 rz 180 deg; joints [-145.866, -85.303, -25.018, 62.875, 39.085, -56.576]
  Call Extruder(269.02049)
  MoveL 3762 to (232.62, 162.8, 59.84) mm, rotated rx 180 ry 0 rz -180 deg; joints [-145.845, -85.271, -25.083, 62.857, 39.117, -56.544]
  MoveL 3763 to (232.62, 162.8, 59.84) mm, rotated rx 180 ry 0 rz -180 deg; joints [-145.845, -85.271, -25.083, 62.857, 39.117, -56.544]
  Call Extruder(269.17786)
  MoveL 3764 to (232.37, 162.91, 59.84) mm, rotated rx 180 ry 0 rz 180 deg; joints [-145.825, -85.24, -25.147, 62.839, 39.149, -56.511]
  MoveL 3765 to (232.37, 162.91, 59.84) mm, rotated rx 180 ry 0 rz 180 deg; joints [-145.825, -85.24, -25.147, 62.839, 39.149, -56.511]
  Call Extruder(269.36060)
  MoveL 3766 to (232.07, 163.02, 59.84) mm, rotated rx -180 ry 0 rz 180 deg; joints [-145.801, -85.202, -25.224, 62.817, 39.187, -56.472]
  MoveL 3767 to (232.07, 163.02, 59.84) mm, rotated rx -180 ry 0 rz 180 deg; joints [-145.801, -85.202, -25.224, 62.817, 39.187, -56.472]
  Call Extruder(269.54259)
  MoveL 3768 to (231.78, 163.15, 59.84) mm, rotated rx -180 ry 0 rz 180 deg; joints [-145.777, -85.165, -25.3, 62.795, 39.225, -56.434]
  MoveL 3769 to (231.78, 163.15, 59.84) mm, rotated rx -180 ry 0 rz 180 deg; joints [-145.777, -85.165, -25.3, 62.795, 39.225, -56.434]
  Call Extruder(269.68992)
  MoveL 3770 to (231.54, 163.24, 59.84) mm, rotated rx -180 ry 0 rz -180 deg; joints [-145.759, -85.133, -25.365, 62.776, 39.255, -56.4]
  MoveL 3771 to (231.54, 163.24, 59.84) mm, rotated rx -180 ry 0 rz -180 deg; joints [-145.759, -85.133, -25.365, 62.776, 39.255, -56.4]
  Call Extruder(269.80315)
  MoveL 3772 to (231.35, 163.3, 59.84) mm, rotated rx 180 ry 0 rz 180 deg; joints [-145.744, -85.107, -25.418, 62.759, 39.28, -56.371]
  MoveL 3773 to (231.35, 163.3, 59.84) mm, rotated rx 180 ry 0 rz 180 deg; joints [-145.744, -85.107, -25.418, 62.759, 39.28, -56.371]
  Call Extruder(269.91592)
  MoveL 3774 to (231.17, 163.36, 59.84) mm, rotated rx 180 ry 0 rz 180 deg; joints [-145.73, -85.081, -25.471, 62.741, 39.304, -56.343]
  MoveL 3775 to (231.17, 163.36, 59.84) mm, rotated rx 180 ry 0 rz 180 deg; joints [-145.73, -85.081, -25.471, 62.741, 39.304, -56.343]
  Call Extruder(270.02826)
  MoveL 3776 to (230.98, 163.42, 59.84) mm, rotated rx 180 ry 0 rz 180 deg; joints [-145.716, -85.055, -25.524, 62.724, 39.328, -56.314]
  MoveL 3777 to (230.98, 163.42, 59.84) mm, rotated rx 180 ry 0 rz 180 deg; joints [-145.716, -85.055, -25.524, 62.724, 39.328, -56.314]
  Call Extruder(270.14014)
  MoveL 3778 to (230.79, 163.48, 59.84) mm, rotated rx -180 ry 0 rz 180 deg; joints [-145.702, -85.03, -25.577, 62.707, 39.352, -56.286]
  MoveL 3779 to (230.79, 163.48, 59.84) mm, rotated rx -180 ry 0 rz 180 deg; joints [-145.702, -85.03, -25.577, 62.707, 39.352, -56.286]
  Call Extruder(270.26155)
  MoveL 3780 to (230.58, 163.55, 59.84) mm, rotated rx -180 ry 0 rz 180 deg; joints [-145.687, -85.001, -25.635, 62.689, 39.378, -56.255]
  MoveL 3781 to (230.58, 163.55, 59.84) mm, rotated rx -180 ry 0 rz 180 deg; joints [-145.687, -85.001, -25.635, 62.689, 39.378, -56.255]
  Call Extruder(270.39236)
  MoveL 3782 to (230.36, 163.61, 59.84) mm, rotated rx -180 ry 0 rz 180 deg; joints [-145.67, -84.97, -25.699, 62.668, 39.407, -56.22]
  MoveL 3783 to (230.36, 163.61, 59.84) mm, rotated rx -180 ry 0 rz 180 deg; joints [-145.67, -84.97, -25.699, 62.668, 39.407, -56.22]
  Call Extruder(270.52261)
  MoveL 3784 to (230.14, 163.68, 59.84) mm, rotated rx -180 ry 0 rz 180 deg; joints [-145.654, -84.939, -25.762, 62.647, 39.436, -56.186]
  MoveL 3785 to (230.14, 163.68, 59.84) mm, rotated rx -180 ry 0 rz 180 deg; joints [-145.654, -84.939, -25.762, 62.647, 39.436, -56.186]
  Call Extruder(270.65229)
  MoveL 3786 to (229.91, 163.75, 59.84) mm, rotated rx 180 ry 0 rz 180 deg; joints [-145.638, -84.908, -25.826, 62.626, 39.464, -56.151]
  MoveL 3787 to (229.91, 163.75, 59.84) mm, rotated rx 180 ry 0 rz 180 deg; joints [-145.638, -84.908, -25.826, 62.626, 39.464, -56.151]
  Call Extruder(270.78141)
  MoveL 3788 to (229.69, 163.82, 59.84) mm, rotated rx 180 ry 0 rz 180 deg; joints [-145.621, -84.877, -25.89, 62.605, 39.493, -56.117]
  MoveL 3789 to (229.69, 163.82, 59.84) mm, rotated rx 180 ry 0 rz 180 deg; joints [-145.621, -84.877, -25.89, 62.605, 39.493, -56.117]
  Call Extruder(270.89648)
  MoveL 3790 to (229.48, 163.86, 59.84) mm, rotated rx -180 ry 0 rz 180 deg; joints [-145.607, -84.847, -25.951, 62.583, 39.519, -56.082]
  MoveL 3791 to (229.48, 163.86, 59.84) mm, rotated rx -180 ry 0 rz 180 deg; joints [-145.607, -84.847, -25.951, 62.583, 39.519, -56.082]
  Call Extruder(271.01110)
  MoveL 3792 to (229.28, 163.91, 59.84) mm, rotated rx 180 ry 0 rz -180 deg; joints [-145.594, -84.817, -26.013, 62.562, 39.545, -56.047]
  MoveL 3793 to (229.28, 163.91, 59.84) mm, rotated rx 180 ry 0 rz -180 deg; joints [-145.594, -84.817, -26.013, 62.562, 39.545, -56.047]
  Call Extruder(271.12527)
  MoveL 3794 to (229.08, 163.95, 59.84) mm, rotated rx 180 ry 0 rz -180 deg; joints [-145.58, -84.786, -26.075, 62.54, 39.571, -56.013]
  MoveL 3795 to (229.08, 163.95, 59.84) mm, rotated rx 180 ry 0 rz -180 deg; joints [-145.58, -84.786, -26.075, 62.54, 39.571, -56.013]
  Call Extruder(271.23899)
  MoveL 3796 to (228.87, 164, 59.84) mm, rotated rx -180 ry 0 rz 180 deg; joints [-145.566, -84.756, -26.137, 62.518, 39.597, -55.978]
  MoveL 3797 to (228.87, 164, 59.84) mm, rotated rx -180 ry 0 rz 180 deg; joints [-145.566, -84.756, -26.137, 62.518, 39.597, -55.978]
  Call Extruder(271.36441)
  MoveL 3798 to (228.64, 164.04, 59.84) mm, rotated rx 180 ry 0 rz 180 deg; joints [-145.551, -84.723, -26.205, 62.493, 39.625, -55.939]
  MoveL 3799 to (228.64, 164.04, 59.84) mm, rotated rx 180 ry 0 rz 180 deg; joints [-145.551, -84.723, -26.205, 62.493, 39.625, -55.939]
  Call Extruder(271.50139)
  MoveL 3800 to (228.4, 164.09, 59.84) mm, rotated rx -180 ry 0 rz -180 deg; joints [-145.535, -84.686, -26.281, 62.466, 39.657, -55.896]
  MoveL 3801 to (228.4, 164.09, 59.84) mm, rotated rx -180 ry 0 rz -180 deg; joints [-145.535, -84.686, -26.281, 62.466, 39.657, -55.896]
  Call Extruder(271.63776)
  MoveL 3802 to (228.15, 164.14, 59.84) mm, rotated rx 180 ry 0 rz 180 deg; joints [-145.518, -84.649, -26.357, 62.439, 39.689, -55.853]
  MoveL 3803 to (228.15, 164.14, 59.84) mm, rotated rx 180 ry 0 rz 180 deg; joints [-145.518, -84.649, -26.357, 62.439, 39.689, -55.853]
  Call Extruder(271.77351)
  MoveL 3804 to (227.9, 164.19, 59.84) mm, rotated rx 180 ry 0 rz 180 deg; joints [-145.502, -84.612, -26.433, 62.412, 39.72, -55.81]
  MoveL 3805 to (227.9, 164.19, 59.84) mm, rotated rx 180 ry 0 rz 180 deg; joints [-145.502, -84.612, -26.433, 62.412, 39.72, -55.81]
  Call Extruder(271.90866)
  MoveL 3806 to (227.65, 164.24, 59.84) mm, rotated rx -180 ry 0 rz 180 deg; joints [-145.485, -84.575, -26.509, 62.385, 39.752, -55.768]
  MoveL 3807 to (227.65, 164.24, 59.84) mm, rotated rx -180 ry 0 rz 180 deg; joints [-145.485, -84.575, -26.509, 62.385, 39.752, -55.768]
  Call Extruder(272.04320)
  MoveL 3808 to (227.4, 164.29, 59.84) mm, rotated rx -180 ry 0 rz 180 deg; joints [-145.469, -84.538, -26.584, 62.358, 39.783, -55.726]
  MoveL 3809 to (227.4, 164.29, 59.84) mm, rotated rx -180 ry 0 rz 180 deg; joints [-145.469, -84.538, -26.584, 62.358, 39.783, -55.726]
  Call Extruder(272.17712)
  MoveL 3810 to (227.15, 164.34, 59.84) mm, rotated rx 180 ry 0 rz 180 deg; joints [-145.453, -84.502, -26.659, 62.332, 39.815, -55.683]
  MoveL 3811 to (227.15, 164.34, 59.84) mm, rotated rx 180 ry 0 rz 180 deg; joints [-145.453, -84.502, -26.659, 62.332, 39.815, -55.683]
  Call Extruder(272.32499)
  MoveL 3812 to (226.87, 164.39, 59.84) mm, rotated rx 180 ry 0 rz -180 deg; joints [-145.435, -84.46, -26.744, 62.301, 39.85, -55.635]
  MoveL 3813 to (226.87, 164.39, 59.84) mm, rotated rx 180 ry 0 rz -180 deg; joints [-145.435, -84.46, -26.744, 62.301, 39.85, -55.635]
  Call Extruder(272.48673)
  MoveL 3814 to (226.57, 164.44, 59.84) mm, rotated rx 180 ry 0 rz 180 deg; joints [-145.415, -84.414, -26.839, 62.267, 39.888, -55.581]
  MoveL 3815 to (226.57, 164.44, 59.84) mm, rotated rx 180 ry 0 rz 180 deg; joints [-145.415, -84.414, -26.839, 62.267, 39.888, -55.581]
  Call Extruder(272.64774)
  MoveL 3816 to (226.26, 164.49, 59.84) mm, rotated rx 180 ry 0 rz -180 deg; joints [-145.396, -84.368, -26.934, 62.232, 39.927, -55.527]
  MoveL 3817 to (226.26, 164.49, 59.84) mm, rotated rx 180 ry 0 rz -180 deg; joints [-145.396, -84.368, -26.934, 62.232, 39.927, -55.527]
  Call Extruder(272.80803)
  MoveL 3818 to (225.96, 164.53, 59.84) mm, rotated rx 180 ry 0 rz 180 deg; joints [-145.377, -84.322, -27.028, 62.198, 39.965, -55.473]
  MoveL 3819 to (225.96, 164.53, 59.84) mm, rotated rx 180 ry 0 rz 180 deg; joints [-145.377, -84.322, -27.028, 62.198, 39.965, -55.473]
  Call Extruder(272.96758)
  MoveL 3820 to (225.65, 164.58, 59.84) mm, rotated rx -180 ry 0 rz 180 deg; joints [-145.357, -84.276, -27.122, 62.165, 40.004, -55.42]
  MoveL 3821 to (225.65, 164.58, 59.84) mm, rotated rx -180 ry 0 rz 180 deg; joints [-145.357, -84.276, -27.122, 62.165, 40.004, -55.42]
  Call Extruder(273.12641)
  MoveL 3822 to (225.34, 164.63, 59.84) mm, rotated rx -180 ry 0 rz 180 deg; joints [-145.338, -84.231, -27.216, 62.131, 40.042, -55.367]
  MoveL 3823 to (225.34, 164.63, 59.84) mm, rotated rx -180 ry 0 rz 180 deg; joints [-145.338, -84.231, -27.216, 62.131, 40.042, -55.367]
  Call Extruder(273.30508)
  MoveL 3824 to (225, 164.68, 59.84) mm, rotated rx 180 ry 0 rz 180 deg; joints [-145.317, -84.178, -27.324, 62.092, 40.086, -55.305]
  MoveL 3825 to (225, 164.68, 59.84) mm, rotated rx 180 ry 0 rz 180 deg; joints [-145.317, -84.178, -27.324, 62.092, 40.086, -55.305]
  Call Extruder(273.50353)
  MoveL 3826 to (224.61, 164.72, 59.84) mm, rotated rx 180 ry 0 rz 180 deg; joints [-145.293, -84.119, -27.445, 62.047, 40.134, -55.235]
  MoveL 3827 to (224.61, 164.72, 59.84) mm, rotated rx 180 ry 0 rz 180 deg; joints [-145.293, -84.119, -27.445, 62.047, 40.134, -55.235]
  Call Extruder(273.70110)
  MoveL 3828 to (224.22, 164.77, 59.84) mm, rotated rx 180 ry 0 rz 180 deg; joints [-145.27, -84.06, -27.567, 62.002, 40.183, -55.166]
  MoveL 3829 to (224.22, 164.77, 59.84) mm, rotated rx 180 ry 0 rz 180 deg; joints [-145.27, -84.06, -27.567, 62.002, 40.183, -55.166]
  Call Extruder(273.89781)
  MoveL 3830 to (223.83, 164.82, 59.84) mm, rotated rx 180 ry 0 rz 180 deg; joints [-145.246, -84.001, -27.688, 61.958, 40.231, -55.097]
  MoveL 3831 to (223.83, 164.82, 59.84) mm, rotated rx 180 ry 0 rz 180 deg; joints [-145.246, -84.001, -27.688, 61.958, 40.231, -55.097]
  Call Extruder(274.09365)
  MoveL 3832 to (223.45, 164.86, 59.84) mm, rotated rx -180 ry 0 rz 180 deg; joints [-145.223, -83.942, -27.809, 61.914, 40.28, -55.027]
  MoveL 3833 to (223.45, 164.86, 59.84) mm, rotated rx -180 ry 0 rz 180 deg; joints [-145.223, -83.942, -27.809, 61.914, 40.28, -55.027]
  Call Extruder(274.38900)
  MoveL 3834 to (222.86, 164.91, 59.84) mm, rotated rx 180 ry 0 rz 180 deg; joints [-145.189, -83.851, -27.997, 61.843, 40.353, -54.919]
  MoveL 3835 to (222.86, 164.91, 59.84) mm, rotated rx 180 ry 0 rz 180 deg; joints [-145.189, -83.851, -27.997, 61.843, 40.353, -54.919]
  Call Extruder(274.68303)
  MoveL 3836 to (222.27, 164.96, 59.84) mm, rotated rx 180 ry 0 rz 180 deg; joints [-145.155, -83.76, -28.184, 61.774, 40.427, -54.81]
  MoveL 3837 to (222.27, 164.96, 59.84) mm, rotated rx 180 ry 0 rz 180 deg; joints [-145.155, -83.76, -28.184, 61.774, 40.427, -54.81]
  Call Extruder(274.97572)
  MoveL 3838 to (221.68, 165, 59.84) mm, rotated rx -180 ry 0 rz 180 deg; joints [-145.121, -83.67, -28.371, 61.705, 40.5, -54.703]
  MoveL 3839 to (221.68, 165, 59.84) mm, rotated rx -180 ry 0 rz 180 deg; joints [-145.121, -83.67, -28.371, 61.705, 40.5, -54.703]
  Call Extruder(275.54917)
  MoveL 3840 to (220.52, 165.05, 59.84) mm, rotated rx -180 ry 0 rz 180 deg; joints [-145.056, -83.487, -28.747, 61.563, 40.644, -54.485]
  MoveL 3841 to (220.52, 165.05, 59.84) mm, rotated rx -180 ry 0 rz 180 deg; joints [-145.056, -83.487, -28.747, 61.563, 40.644, -54.485]
  Call Extruder(276.26318)
  MoveL 3842 to (219.06, 165.09, 59.84) mm, rotated rx 180 ry 0 rz -180 deg; joints [-144.977, -83.26, -29.216, 61.387, 40.824, -54.212]
  Call Extruder(393.10992)
  MoveL 3843 to (-19.06, 165.09, 59.84) mm, rotated rx 180 ry 0 rz -180 deg; joints [-127.435, -62.882, -75.214, 60.328, 66.047, -35.473]
  Call Extruder(393.53852)
  MoveL 3844 to (-19.94, 165.07, 59.84) mm, rotated rx -180 ry 0 rz 180 deg; joints [-127.348, -62.84, -75.323, 60.379, 66.131, -35.44]
  MoveL 3845 to (-19.94, 165.07, 59.84) mm, rotated rx -180 ry 0 rz 180 deg; joints [-127.348, -62.84, -75.323, 60.379, 66.131, -35.44]
  Call Extruder(394.11197)
  MoveL 3846 to (-21.1, 165.02, 59.84) mm, rotated rx 180 ry 0 rz -180 deg; joints [-127.235, -62.783, -75.47, 60.446, 66.241, -35.395]
  MoveL 3847 to (-21.1, 165.02, 59.84) mm, rotated rx 180 ry 0 rz -180 deg; joints [-127.235, -62.783, -75.47, 60.446, 66.241, -35.395]
  Call Extruder(394.54627)
  MoveL 3848 to (-21.97, 164.98, 59.84) mm, rotated rx 180 ry 0 rz -180 deg; joints [-127.15, -62.739, -75.583, 60.495, 66.325, -35.359]
  MoveL 3849 to (-21.97, 164.98, 59.84) mm, rotated rx 180 ry 0 rz -180 deg; joints [-127.15, -62.739, -75.583, 60.495, 66.325, -35.359]
  Call Extruder(394.84030)
  MoveL 3850 to (-22.56, 164.93, 59.84) mm, rotated rx 180 ry 0 rz 180 deg; joints [-127.093, -62.709, -75.662, 60.526, 66.381, -35.333]
  MoveL 3851 to (-22.56, 164.93, 59.84) mm, rotated rx 180 ry 0 rz 180 deg; joints [-127.093, -62.709, -75.662, 60.526, 66.381, -35.333]
  Call Extruder(395.13566)
  MoveL 3852 to (-23.15, 164.89, 59.84) mm, rotated rx 180 ry 0 rz 180 deg; joints [-127.037, -62.679, -75.74, 60.558, 66.437, -35.307]
  MoveL 3853 to (-23.15, 164.89, 59.84) mm, rotated rx 180 ry 0 rz 180 deg; joints [-127.037, -62.679, -75.74, 60.558, 66.437, -35.307]
  Call Extruder(395.38188)
  MoveL 3854 to (-23.64, 164.84, 59.84) mm, rotated rx -180 ry 0 rz -180 deg; joints [-126.991, -62.654, -75.806, 60.584, 66.484, -35.285]
  MoveL 3855 to (-23.64, 164.84, 59.84) mm, rotated rx -180 ry 0 rz -180 deg; joints [-126.991, -62.654, -75.806, 60.584, 66.484, -35.285]
  Call Extruder(395.57858)
  MoveL 3856 to (-24.03, 164.79, 59.84) mm, rotated rx 180 ry 0 rz -180 deg; joints [-126.955, -62.634, -75.859, 60.603, 66.521, -35.267]
  MoveL 3857 to (-24.03, 164.79, 59.84) mm, rotated rx 180 ry 0 rz -180 deg; joints [-126.955, -62.634, -75.859, 60.603, 66.521, -35.267]
  Call Extruder(395.77616)
  MoveL 3858 to (-24.42, 164.75, 59.84) mm, rotated rx 180 ry 0 rz 180 deg; joints [-126.919, -62.613, -75.913, 60.622, 66.558, -35.248]
  MoveL 3859 to (-24.42, 164.75, 59.84) mm, rotated rx 180 ry 0 rz 180 deg; joints [-126.919, -62.613, -75.913, 60.622, 66.558, -35.248]
  Call Extruder(395.97460)
  MoveL 3860 to (-24.8, 164.7, 59.84) mm, rotated rx 180 ry 0 rz 180 deg; joints [-126.883, -62.593, -75.966, 60.642, 66.595, -35.229]
  MoveL 3861 to (-24.8, 164.7, 59.84) mm, rotated rx 180 ry 0 rz 180 deg; joints [-126.883, -62.593, -75.966, 60.642, 66.595, -35.229]
  Call Extruder(396.17391)
  MoveL 3862 to (-25.19, 164.66, 59.84) mm, rotated rx -180 ry 0 rz 180 deg; joints [-126.847, -62.572, -76.02, 60.662, 66.632, -35.211]
  MoveL 3863 to (-25.19, 164.66, 59.84) mm, rotated rx -180 ry 0 rz 180 deg; joints [-126.847, -62.572, -76.02, 60.662, 66.632, -35.211]
  Call Extruder(396.33274)
  MoveL 3864 to (-25.5, 164.61, 59.84) mm, rotated rx 180 ry 0 rz 180 deg; joints [-126.82, -62.556, -76.064, 60.676, 66.661, -35.194]
  MoveL 3865 to (-25.5, 164.61, 59.84) mm, rotated rx 180 ry 0 rz 180 deg; joints [-126.82, -62.556, -76.064, 60.676, 66.661, -35.194]
  Call Extruder(396.49230)
  MoveL 3866 to (-25.8, 164.56, 59.84) mm, rotated rx 180 ry 0 rz -180 deg; joints [-126.792, -62.539, -76.108, 60.69, 66.69, -35.178]
  MoveL 3867 to (-25.8, 164.56, 59.84) mm, rotated rx 180 ry 0 rz -180 deg; joints [-126.792, -62.539, -76.108, 60.69, 66.69, -35.178]
  Call Extruder(396.65259)
  MoveL 3868 to (-26.11, 164.51, 59.84) mm, rotated rx 180 ry 0 rz 180 deg; joints [-126.765, -62.522, -76.152, 60.704, 66.719, -35.162]
  MoveL 3869 to (-26.11, 164.51, 59.84) mm, rotated rx 180 ry 0 rz 180 deg; joints [-126.765, -62.522, -76.152, 60.704, 66.719, -35.162]
  Call Extruder(396.81360)
  MoveL 3870 to (-26.41, 164.46, 59.84) mm, rotated rx 180 ry 0 rz 180 deg; joints [-126.737, -62.505, -76.196, 60.719, 66.748, -35.146]
  MoveL 3871 to (-26.41, 164.46, 59.84) mm, rotated rx 180 ry 0 rz 180 deg; joints [-126.737, -62.505, -76.196, 60.719, 66.748, -35.146]
  Call Extruder(396.97535)
  MoveL 3872 to (-26.72, 164.41, 59.84) mm, rotated rx -180 ry 0 rz -180 deg; joints [-126.71, -62.488, -76.24, 60.733, 66.778, -35.13]
  MoveL 3873 to (-26.72, 164.41, 59.84) mm, rotated rx -180 ry 0 rz -180 deg; joints [-126.71, -62.488, -76.24, 60.733, 66.778, -35.13]
  Call Extruder(397.13782)
  MoveL 3874 to (-27.03, 164.36, 59.84) mm, rotated rx -180 ry 0 rz 180 deg; joints [-126.682, -62.472, -76.284, 60.748, 66.807, -35.114]
  MoveL 3875 to (-27.03, 164.36, 59.84) mm, rotated rx -180 ry 0 rz 180 deg; joints [-126.682, -62.472, -76.284, 60.748, 66.807, -35.114]
  Call Extruder(397.27175)
  MoveL 3876 to (-27.27, 164.32, 59.84) mm, rotated rx -180 ry 0 rz 180 deg; joints [-126.66, -62.457, -76.321, 60.758, 66.831, -35.1]
  MoveL 3877 to (-27.27, 164.32, 59.84) mm, rotated rx -180 ry 0 rz 180 deg; joints [-126.66, -62.457, -76.321, 60.758, 66.831, -35.1]
  Call Extruder(397.40628)
  MoveL 3878 to (-27.52, 164.27, 59.84) mm, rotated rx 180 ry 0 rz 180 deg; joints [-126.638, -62.443, -76.358, 60.769, 66.854, -35.085]
  MoveL 3879 to (-27.52, 164.27, 59.84) mm, rotated rx 180 ry 0 rz 180 deg; joints [-126.638, -62.443, -76.358, 60.769, 66.854, -35.085]
  Call Extruder(397.54143)
  MoveL 3880 to (-27.77, 164.22, 59.84) mm, rotated rx -180 ry 0 rz 180 deg; joints [-126.617, -62.429, -76.395, 60.78, 66.878, -35.071]
  MoveL 3881 to (-27.77, 164.22, 59.84) mm, rotated rx -180 ry 0 rz 180 deg; joints [-126.617, -62.429, -76.395, 60.78, 66.878, -35.071]
  Call Extruder(397.67719)
  MoveL 3882 to (-28.02, 164.17, 59.84) mm, rotated rx 180 ry 0 rz -180 deg; joints [-126.595, -62.415, -76.433, 60.791, 66.902, -35.057]
  MoveL 3883 to (-28.02, 164.17, 59.84) mm, rotated rx 180 ry 0 rz -180 deg; joints [-126.595, -62.415, -76.433, 60.791, 66.902, -35.057]
  Call Extruder(397.81355)
  MoveL 3884 to (-28.27, 164.12, 59.84) mm, rotated rx 180 ry 0 rz 180 deg; joints [-126.573, -62.401, -76.47, 60.802, 66.926, -35.043]
  MoveL 3885 to (-28.27, 164.12, 59.84) mm, rotated rx 180 ry 0 rz 180 deg; joints [-126.573, -62.401, -76.47, 60.802, 66.926, -35.043]
  Call Extruder(397.89841)
  MoveL 3886 to (-28.43, 164.09, 59.84) mm, rotated rx 180 ry 0 rz -180 deg; joints [-126.559, -62.392, -76.493, 60.808, 66.94, -35.034]
  Set speed (130.0 mm/s)
  MoveL 3887 to (-31.76, 163.31, 59.84) mm, rotated rx 180 ry 0 rz 180 deg; joints [-126.274, -62.197, -77.006, 60.945, 67.259, -34.83]
  MoveL 3888 to (-31.76, 163.31, 69.25) mm, rotated rx 180 ry 0 rz 180 deg; joints [-126.274, -60.901, -77.684, 61.173, 66.959, -35.418]
  Call Extruder(395.89841)
  Set speed (40.0 mm/s)
  MoveL 3889 to (-31.76, 163.31, 69.25) mm, rotated rx 180 ry 0 rz 180 deg; joints [-126.274, -60.901, -77.684, 61.173, 66.959, -35.418]
  Call Extruder(0.00000)
  Set speed (130.0 mm/s)
  MoveL 3890 to (-31.64, 163.21, 69.25) mm, rotated rx -180 ry 0 rz -180 deg; joints [-126.294, -60.9, -77.686, 61.155, 66.948, -35.41]
  Call Extruder(2.00000)
  Set speed (40.0 mm/s)
  MoveL 3891 to (-31.64, 163.21, 69.25) mm, rotated rx -180 ry 0 rz -180 deg; joints [-126.294, -60.9, -77.686, 61.155, 66.948, -35.41]
  Set speed (30.0 mm/s)
  MoveL 3892 to (-31.64, 163.21, 69.25) mm, rotated rx -180 ry 0 rz -180 deg; joints [-126.294, -60.9, -77.686, 61.155, 66.948, -35.41]
  Call Extruder(2.18198)
  MoveL 3893 to (-31.93, 163.09, 69.25) mm, rotated rx -180 ry 0 rz 180 deg; joints [-126.273, -60.88, -77.739, 61.162, 66.976, -35.386]
  MoveL 3894 to (-31.93, 163.09, 69.25) mm, rotated rx -180 ry 0 rz 180 deg; joints [-126.273, -60.88, -77.739, 61.162, 66.976, -35.386]
  Call Extruder(2.36471)
  MoveL 3895 to (-32.22, 162.97, 69.25) mm, rotated rx -180 ry 0 rz 180 deg; joints [-126.252, -60.859, -77.792, 61.168, 67.004, -35.363]
  MoveL 3896 to (-32.22, 162.97, 69.25) mm, rotated rx -180 ry 0 rz 180 deg; joints [-126.252, -60.859, -77.792, 61.168, 67.004, -35.363]
  Call Extruder(2.53513)
  MoveL 3897 to (-32.49, 162.85, 69.25) mm, rotated rx 180 ry 0 rz 180 deg; joints [-126.233, -60.84, -77.841, 61.174, 67.03, -35.341]
  MoveL 3898 to (-32.49, 162.85, 69.25) mm, rotated rx 180 ry 0 rz 180 deg; joints [-126.233, -60.84, -77.841, 61.174, 67.03, -35.341]
  Call Extruder(2.69310)
  MoveL 3899 to (-32.74, 162.74, 69.25) mm, rotated rx -180 ry 0 rz 180 deg; joints [-126.215, -60.822, -77.887, 61.18, 67.054, -35.32]
  MoveL 3900 to (-32.74, 162.74, 69.25) mm, rotated rx -180 ry 0 rz 180 deg; joints [-126.215, -60.822, -77.887, 61.18, 67.054, -35.32]
  Call Extruder(2.85168)
  MoveL 3901 to (-32.99, 162.64, 69.25) mm, rotated rx -180 ry 0 rz -180 deg; joints [-126.197, -60.805, -77.933, 61.185, 67.078, -35.299]
  MoveL 3902 to (-32.99, 162.64, 69.25) mm, rotated rx -180 ry 0 rz -180 deg; joints [-126.197, -60.805, -77.933, 61.185, 67.078, -35.299]
  Call Extruder(3.05784)
  MoveL 3903 to (-33.29, 162.46, 69.25) mm, rotated rx 180 ry 0 rz 180 deg; joints [-126.179, -60.781, -77.996, 61.187, 67.107, -35.269]
  MoveL 3904 to (-33.29, 162.46, 69.25) mm, rotated rx 180 ry 0 rz 180 deg; joints [-126.179, -60.781, -77.996, 61.187, 67.107, -35.269]
  Call Extruder(3.26479)
  MoveL 3905 to (-33.6, 162.29, 69.25) mm, rotated rx -180 ry 0 rz 180 deg; joints [-126.16, -60.756, -78.059, 61.189, 67.136, -35.238]
  MoveL 3906 to (-33.6, 162.29, 69.25) mm, rotated rx -180 ry 0 rz 180 deg; joints [-126.16, -60.756, -78.059, 61.189, 67.136, -35.238]
  Call Extruder(3.47251)
  MoveL 3907 to (-33.9, 162.11, 69.25) mm, rotated rx 180 ry 0 rz 180 deg; joints [-126.142, -60.732, -78.122, 61.191, 67.166, -35.208]
  MoveL 3908 to (-33.9, 162.11, 69.25) mm, rotated rx 180 ry 0 rz 180 deg; joints [-126.142, -60.732, -78.122, 61.191, 67.166, -35.208]
  Call Extruder(3.68101)
  MoveL 3909 to (-34.21, 161.94, 69.25) mm, rotated rx 180 ry 0 rz -180 deg; joints [-126.123, -60.708, -78.184, 61.193, 67.195, -35.177]
  MoveL 3910 to (-34.21, 161.94, 69.25) mm, rotated rx 180 ry 0 rz -180 deg; joints [-126.123, -60.708, -78.184, 61.193, 67.195, -35.177]
  Call Extruder(3.86055)
  MoveL 3911 to (-34.45, 161.76, 69.25) mm, rotated rx 180 ry 0 rz 180 deg; joints [-126.111, -60.687, -78.24, 61.191, 67.218, -35.149]
  MoveL 3912 to (-34.45, 161.76, 69.25) mm, rotated rx 180 ry 0 rz 180 deg; joints [-126.111, -60.687, -78.24, 61.191, 67.218, -35.149]
  Call Extruder(4.19399)
  MoveL 3913 to (-34.9, 161.43, 69.25) mm, rotated rx -180 ry 0 rz -180 deg; joints [-126.089, -60.647, -78.344, 61.187, 67.262, -35.096]
  MoveL 3914 to (-34.9, 161.43, 69.25) mm, rotated rx -180 ry 0 rz -180 deg; joints [-126.089, -60.647, -78.344, 61.187, 67.262, -35.096]
  Call Extruder(4.52861)
  MoveL 3915 to (-35.35, 161.1, 69.25) mm, rotated rx 180 ry 0 rz 180 deg; joints [-126.067, -60.607, -78.448, 61.184, 67.306, -35.043]
  Call Extruder(5.35652)
  MoveL 3916 to (-36.39, 160.19, 69.25) mm, rotated rx -180 ry 0 rz -180 deg; joints [-126.027, -60.507, -78.71, 61.159, 67.406, -34.902]
  Call Extruder(5.98652)
  MoveL 3917 to (-37.09, 159.4, 69.25) mm, rotated rx 180 ry 0 rz 180 deg; joints [-126.014, -60.429, -78.914, 61.125, 67.475, -34.787]
  Call Extruder(6.31951)
  MoveL 3918 to (-37.44, 158.97, 69.25) mm, rotated rx 180 ry 0 rz 180 deg; joints [-126.011, -60.388, -79.021, 61.104, 67.509, -34.725]
  MoveL 3919 to (-37.44, 158.97, 69.25) mm, rotated rx 180 ry 0 rz 180 deg; joints [-126.011, -60.388, -79.021, 61.104, 67.509, -34.725]
  Call Extruder(6.58931)
  MoveL 3920 to (-37.7, 158.61, 69.25) mm, rotated rx 180 ry 0 rz 180 deg; joints [-126.011, -60.355, -79.109, 61.085, 67.535, -34.674]
  Set speed (130.0 mm/s)
  MoveL 3921 to (-37.7, 158.61, 69.25) mm, rotated rx 180 ry 0 rz 180 deg; joints [-126.011, -60.355, -79.109, 61.085, 67.535, -34.674]
  Set speed (30.0 mm/s)
  MoveL 3922 to (-37.7, 158.61, 69.25) mm, rotated rx 180 ry 0 rz 180 deg; joints [-126.011, -60.355, -79.109, 61.085, 67.535, -34.674]
  Call Extruder(6.87472)
  MoveL 3923 to (-37.98, 158.22, 69.25) mm, rotated rx 180 ry 0 rz 180 deg; joints [-126.011, -60.319, -79.202, 61.064, 67.563, -34.62]
  MoveL 3924 to (-37.98, 158.22, 69.25) mm, rotated rx 180 ry 0 rz 180 deg; joints [-126.011, -60.319, -79.202, 61.064, 67.563, -34.62]
  Call Extruder(7.13432)
  MoveL 3925 to (-38.22, 157.85, 69.25) mm, rotated rx 180 ry 0 rz 180 deg; joints [-126.013, -60.287, -79.286, 61.042, 67.587, -34.569]
  MoveL 3926 to (-38.22, 157.85, 69.25) mm, rotated rx 180 ry 0 rz 180 deg; joints [-126.013, -60.287, -79.286, 61.042, 67.587, -34.569]
  Call Extruder(7.34204)
  MoveL 3927 to (-38.4, 157.55, 69.25) mm, rotated rx 180 ry 0 rz 180 deg; joints [-126.018, -60.262, -79.354, 61.023, 67.604, -34.528]
  MoveL 3928 to (-38.4, 157.55, 69.25) mm, rotated rx 180 ry 0 rz 180 deg; joints [-126.018, -60.262, -79.354, 61.023, 67.604, -34.528]
  Call Extruder(7.54898)
  MoveL 3929 to (-38.57, 157.25, 69.25) mm, rotated rx -180 ry 0 rz 180 deg; joints [-126.023, -60.236, -79.421, 61.004, 67.622, -34.487]
  MoveL 3930 to (-38.57, 157.25, 69.25) mm, rotated rx -180 ry 0 rz 180 deg; joints [-126.023, -60.236, -79.421, 61.004, 67.622, -34.487]
  Call Extruder(7.75514)
  MoveL 3931 to (-38.75, 156.94, 69.25) mm, rotated rx 180 ry 0 rz 180 deg; joints [-126.028, -60.211, -79.488, 60.984, 67.639, -34.445]
  MoveL 3932 to (-38.75, 156.94, 69.25) mm, rotated rx 180 ry 0 rz 180 deg; joints [-126.028, -60.211, -79.488, 60.984, 67.639, -34.445]
  Call Extruder(7.93681)
  MoveL 3933 to (-38.89, 156.66, 69.25) mm, rotated rx 180 ry 0 rz -180 deg; joints [-126.034, -60.188, -79.548, 60.965, 67.654, -34.408]
  MoveL 3934 to (-38.89, 156.66, 69.25) mm, rotated rx 180 ry 0 rz -180 deg; joints [-126.034, -60.188, -79.548, 60.965, 67.654, -34.408]
  Call Extruder(8.09480)
  MoveL 3935 to (-39, 156.42, 69.25) mm, rotated rx -180 ry 0 rz 180 deg; joints [-126.042, -60.169, -79.599, 60.947, 67.665, -34.376]
  MoveL 3936 to (-39, 156.42, 69.25) mm, rotated rx -180 ry 0 rz 180 deg; joints [-126.042, -60.169, -79.599, 60.947, 67.665, -34.376]
  Call Extruder(8.25218)
  MoveL 3937 to (-39.1, 156.17, 69.25) mm, rotated rx 180 ry 0 rz 180 deg; joints [-126.05, -60.149, -79.65, 60.928, 67.675, -34.343]
  MoveL 3938 to (-39.1, 156.17, 69.25) mm, rotated rx 180 ry 0 rz 180 deg; joints [-126.05, -60.149, -79.65, 60.928, 67.675, -34.343]
  Call Extruder(8.43490)
  MoveL 3939 to (-39.23, 155.88, 69.25) mm, rotated rx 180 ry 0 rz 180 deg; joints [-126.06, -60.127, -79.709, 60.906, 67.688, -34.305]
  MoveL 3940 to (-39.23, 155.88, 69.25) mm, rotated rx 180 ry 0 rz 180 deg; joints [-126.06, -60.127, -79.709, 60.906, 67.688, -34.305]
  Call Extruder(8.61686)
  MoveL 3941 to (-39.35, 155.58, 69.25) mm, rotated rx 180 ry 0 rz 180 deg; joints [-126.07, -60.105, -79.768, 60.884, 67.7, -34.267]
  MoveL 3942 to (-39.35, 155.58, 69.25) mm, rotated rx 180 ry 0 rz 180 deg; joints [-126.07, -60.105, -79.768, 60.884, 67.7, -34.267]
  Call Extruder(8.76420)
  MoveL 3943 to (-39.44, 155.34, 69.25) mm, rotated rx 180 ry 0 rz -180 deg; joints [-126.079, -60.087, -79.816, 60.866, 67.71, -34.236]
  MoveL 3944 to (-39.44, 155.34, 69.25) mm, rotated rx 180 ry 0 rz -180 deg; joints [-126.079, -60.087, -79.816, 60.866, 67.71, -34.236]
  Call Extruder(8.87743)
  MoveL 3945 to (-39.5, 155.15, 69.25) mm, rotated rx 180 ry 0 rz 180 deg; joints [-126.087, -60.073, -79.852, 60.851, 67.716, -34.212]
  MoveL 3946 to (-39.5, 155.15, 69.25) mm, rotated rx 180 ry 0 rz 180 deg; joints [-126.087, -60.073, -79.852, 60.851, 67.716, -34.212]
  Call Extruder(8.99022)
  MoveL 3947 to (-39.56, 154.97, 69.25) mm, rotated rx -180 ry 0 rz -180 deg; joints [-126.095, -60.059, -79.888, 60.835, 67.722, -34.188]
  MoveL 3948 to (-39.56, 154.97, 69.25) mm, rotated rx -180 ry 0 rz -180 deg; joints [-126.095, -60.059, -79.888, 60.835, 67.722, -34.188]
  Call Extruder(9.10257)
  MoveL 3949 to (-39.62, 154.78, 69.25) mm, rotated rx 180 ry 0 rz -180 deg; joints [-126.103, -60.046, -79.925, 60.82, 67.729, -34.164]
  MoveL 3950 to (-39.62, 154.78, 69.25) mm, rotated rx 180 ry 0 rz -180 deg; joints [-126.103, -60.046, -79.925, 60.82, 67.729, -34.164]
  Call Extruder(9.21447)
  MoveL 3951 to (-39.68, 154.59, 69.25) mm, rotated rx 180 ry 0 rz 180 deg; joints [-126.111, -60.032, -79.961, 60.804, 67.735, -34.14]
  MoveL 3952 to (-39.68, 154.59, 69.25) mm, rotated rx 180 ry 0 rz 180 deg; joints [-126.111, -60.032, -79.961, 60.804, 67.735, -34.14]
  Call Extruder(9.33587)
  MoveL 3953 to (-39.75, 154.38, 69.25) mm, rotated rx 180 ry 0 rz 180 deg; joints [-126.12, -60.017, -80, 60.788, 67.742, -34.113]
  MoveL 3954 to (-39.75, 154.38, 69.25) mm, rotated rx 180 ry 0 rz 180 deg; joints [-126.12, -60.017, -80, 60.788, 67.742, -34.113]
  Call Extruder(9.46666)
  MoveL 3955 to (-39.82, 154.16, 69.25) mm, rotated rx 180 ry 0 rz 180 deg; joints [-126.131, -60.001, -80.043, 60.769, 67.749, -34.085]
  MoveL 3956 to (-39.82, 154.16, 69.25) mm, rotated rx 180 ry 0 rz 180 deg; joints [-126.131, -60.001, -80.043, 60.769, 67.749, -34.085]
  Call Extruder(9.59689)
  MoveL 3957 to (-39.88, 153.94, 69.25) mm, rotated rx -180 ry 0 rz 180 deg; joints [-126.141, -59.985, -80.085, 60.75, 67.756, -34.057]
  MoveL 3958 to (-39.88, 153.94, 69.25) mm, rotated rx -180 ry 0 rz 180 deg; joints [-126.141, -59.985, -80.085, 60.75, 67.756, -34.057]
  Call Extruder(9.72656)
  MoveL 3959 to (-39.95, 153.71, 69.25) mm, rotated rx 180 ry 0 rz 180 deg; joints [-126.151, -59.969, -80.127, 60.732, 67.764, -34.028]
  MoveL 3960 to (-39.95, 153.71, 69.25) mm, rotated rx 180 ry 0 rz 180 deg; joints [-126.151, -59.969, -80.127, 60.732, 67.764, -34.028]
  Call Extruder(9.85565)
  MoveL 3961 to (-40.02, 153.49, 69.25) mm, rotated rx -180 ry 0 rz 180 deg; joints [-126.161, -59.953, -80.169, 60.713, 67.771, -34]
  MoveL 3962 to (-40.02, 153.49, 69.25) mm, rotated rx -180 ry 0 rz 180 deg; joints [-126.161, -59.953, -80.169, 60.713, 67.771, -34]
  Call Extruder(9.97074)
  MoveL 3963 to (-40.06, 153.28, 69.25) mm, rotated rx 180 ry 0 rz -180 deg; joints [-126.173, -59.94, -80.206, 60.695, 67.776, -33.975]
  MoveL 3964 to (-40.06, 153.28, 69.25) mm, rotated rx 180 ry 0 rz -180 deg; joints [-126.173, -59.94, -80.206, 60.695, 67.776, -33.975]
  Call Extruder(10.08538)
  MoveL 3965 to (-40.11, 153.08, 69.25) mm, rotated rx 180 ry 0 rz 180 deg; joints [-126.184, -59.926, -80.243, 60.677, 67.781, -33.949]
  MoveL 3966 to (-40.11, 153.08, 69.25) mm, rotated rx 180 ry 0 rz 180 deg; joints [-126.184, -59.926, -80.243, 60.677, 67.781, -33.949]
  Call Extruder(10.19956)
  MoveL 3967 to (-40.15, 152.88, 69.25) mm, rotated rx 180 ry 0 rz -180 deg; joints [-126.195, -59.912, -80.279, 60.659, 67.785, -33.924]
  MoveL 3968 to (-40.15, 152.88, 69.25) mm, rotated rx 180 ry 0 rz -180 deg; joints [-126.195, -59.912, -80.279, 60.659, 67.785, -33.924]
  Call Extruder(10.31329)
  MoveL 3969 to (-40.2, 152.67, 69.25) mm, rotated rx 180 ry 0 rz 180 deg; joints [-126.206, -59.898, -80.316, 60.64, 67.79, -33.899]
  MoveL 3970 to (-40.2, 152.67, 69.25) mm, rotated rx 180 ry 0 rz 180 deg; joints [-126.206, -59.898, -80.316, 60.64, 67.79, -33.899]
  Call Extruder(10.43872)
  MoveL 3971 to (-40.24, 152.45, 69.25) mm, rotated rx 180 ry 0 rz -180 deg; joints [-126.219, -59.883, -80.356, 60.62, 67.796, -33.871]
  MoveL 3972 to (-40.24, 152.45, 69.25) mm, rotated rx 180 ry 0 rz -180 deg; joints [-126.219, -59.883, -80.356, 60.62, 67.796, -33.871]
  Call Extruder(10.57569)
  MoveL 3973 to (-40.29, 152.2, 69.25) mm, rotated rx 180 ry 0 rz 180 deg; joints [-126.233, -59.867, -80.401, 60.597, 67.801, -33.84]
  MoveL 3974 to (-40.29, 152.2, 69.25) mm, rotated rx 180 ry 0 rz 180 deg; joints [-126.233, -59.867, -80.401, 60.597, 67.801, -33.84]
  Call Extruder(10.71206)
  MoveL 3975 to (-40.34, 151.95, 69.25) mm, rotated rx -180 ry 0 rz 180 deg; joints [-126.248, -59.85, -80.445, 60.575, 67.807, -33.809]
  MoveL 3976 to (-40.34, 151.95, 69.25) mm, rotated rx -180 ry 0 rz 180 deg; joints [-126.248, -59.85, -80.445, 60.575, 67.807, -33.809]
  Call Extruder(10.84781)
  MoveL 3977 to (-40.39, 151.7, 69.25) mm, rotated rx 180 ry 0 rz 180 deg; joints [-126.262, -59.833, -80.489, 60.552, 67.812, -33.778]
  MoveL 3978 to (-40.39, 151.7, 69.25) mm, rotated rx 180 ry 0 rz 180 deg; joints [-126.262, -59.833, -80.489, 60.552, 67.812, -33.778]
  Call Extruder(10.98296)
  MoveL 3979 to (-40.44, 151.45, 69.25) mm, rotated rx -180 ry 0 rz -180 deg; joints [-126.276, -59.817, -80.533, 60.529, 67.818, -33.748]
  MoveL 3980 to (-40.44, 151.45, 69.25) mm, rotated rx -180 ry 0 rz -180 deg; joints [-126.276, -59.817, -80.533, 60.529, 67.818, -33.748]
  Call Extruder(11.11749)
  MoveL 3981 to (-40.49, 151.2, 69.25) mm, rotated rx 180 ry 0 rz 180 deg; joints [-126.291, -59.8, -80.577, 60.507, 67.824, -33.717]
  MoveL 3982 to (-40.49, 151.2, 69.25) mm, rotated rx 180 ry 0 rz 180 deg; joints [-126.291, -59.8, -80.577, 60.507, 67.824, -33.717]
  Call Extruder(11.25142)
  MoveL 3983 to (-40.54, 150.95, 69.25) mm, rotated rx 180 ry 0 rz 180 deg; joints [-126.305, -59.784, -80.621, 60.484, 67.829, -33.686]
  MoveL 3984 to (-40.54, 150.95, 69.25) mm, rotated rx 180 ry 0 rz 180 deg; joints [-126.305, -59.784, -80.621, 60.484, 67.829, -33.686]
  Call Extruder(11.39927)
  MoveL 3985 to (-40.59, 150.67, 69.25) mm, rotated rx 180 ry 0 rz -180 deg; joints [-126.322, -59.766, -80.669, 60.458, 67.835, -33.652]
  MoveL 3986 to (-40.59, 150.67, 69.25) mm, rotated rx 180 ry 0 rz -180 deg; joints [-126.322, -59.766, -80.669, 60.458, 67.835, -33.652]
  Call Extruder(11.56100)
  MoveL 3987 to (-40.64, 150.37, 69.25) mm, rotated rx 180 ry 0 rz 180 deg; joints [-126.341, -59.746, -80.721, 60.43, 67.84, -33.615]
  MoveL 3988 to (-40.64, 150.37, 69.25) mm, rotated rx 180 ry 0 rz 180 deg; joints [-126.341, -59.746, -80.721, 60.43, 67.84, -33.615]
  Call Extruder(11.72199)
  MoveL 3989 to (-40.69, 150.06, 69.25) mm, rotated rx 180 ry 0 rz 180 deg; joints [-126.36, -59.727, -80.774, 60.401, 67.846, -33.578]
  MoveL 3990 to (-40.69, 150.06, 69.25) mm, rotated rx 180 ry 0 rz 180 deg; joints [-126.36, -59.727, -80.774, 60.401, 67.846, -33.578]
  Call Extruder(11.88226)
